    LOCAL CONST Robtarget Tr_meulage_bavure_297 := [[34.2176875,132.965375,122.45971875],[0.142128156611238,-0.169112950759258,-0.746628793402951,0.62749170659495],[0,0,0,0],[8.999999E+09,8.999999E+09,8.999999E+09,8.999999E+09,8.999999E+09,8.999999E+09]];
    LOCAL CONST Robtarget Tr_meulage_bavure_298 := [[35.4824296875,132.352796875,122.428859375],[0.141640226442861,-0.168636903428218,-0.74693783228447,0.62736234805536],[0,0,0,0],[8.999999E+09,8.999999E+09,8.999999E+09,8.999999E+09,8.999999E+09,8.999999E+09]];
    LOCAL CONST Robtarget Tr_meulage_bavure_299 := [[38.3330234375,131.063109375,122.374390625],[0.14118721471856,-0.168181992906434,-0.74720342134066,0.627270304413374],[0,0,0,0],[8.999999E+09,8.999999E+09,8.999999E+09,8.999999E+09,8.999999E+09,8.999999E+09]];
    LOCAL CONST Robtarget Tr_meulage_bavure_300 := [[39.25145703125,130.60725,122.35015625],[0.14084665051928,-0.16784433536859,-0.747410861926925,0.627190165417019],[0,0,0,0],[8.999999E+09,8.999999E+09,8.999999E+09,8.999999E+09,8.999999E+09,8.999999E+09]];
    LOCAL CONST Robtarget Tr_meulage_bavure_301 := [[43.699125,128.5305,122.2544765625],[0.140654971334551,-0.167669079521495,-0.747553059163392,0.627110582390972],[0,0,0,0],[8.999999E+09,8.999999E+09,8.999999E+09,8.999999E+09,8.999999E+09,8.999999E+09]];
    LOCAL CONST Robtarget Tr_meulage_bavure_302 := [[44.1365078125,128.3245625,122.24478125],[0.140603570004533,-0.167647641561045,-0.747634929696438,0.62703023553797],[0,0,0,0],[8.999999E+09,8.999999E+09,8.999999E+09,8.999999E+09,8.999999E+09,8.999999E+09]];
    LOCAL CONST Robtarget Tr_meulage_bavure_303 := [[44.23293359375,128.27996875,122.24278125],[0.14065985839217,-0.167741895489389,-0.747666250712567,0.626955052838826],[0,0,0,0],[8.999999E+09,8.999999E+09,8.999999E+09,8.999999E+09,8.999999E+09,8.999999E+09]];
    LOCAL CONST Robtarget Tr_meulage_bavure_304 := [[44.98623046875,127.9280703125,122.226546875],[0.140804799027706,-0.167930767749504,-0.747654793054834,0.626885616548954],[0,0,0,0],[8.999999E+09,8.999999E+09,8.999999E+09,8.999999E+09,8.999999E+09,8.999999E+09]];
    LOCAL CONST Robtarget Tr_meulage_bavure_305 := [[45.85191015625,127.5197578125,122.20725],[0.141050378042018,-0.168230430617468,-0.747600477109053,0.626814836849593],[0,0,0,0],[8.999999E+09,8.999999E+09,8.999999E+09,8.999999E+09,8.999999E+09,8.999999E+09]];
    LOCAL CONST Robtarget Tr_meulage_bavure_306 := [[46.1492265625,127.3825234375,122.2011171875],[0.141429042259318,-0.168679406784711,-0.747494198232892,0.626735596037544],[0,0,0,0],[8.999999E+09,8.999999E+09,8.999999E+09,8.999999E+09,8.999999E+09,8.999999E+09]];
    LOCAL CONST Robtarget Tr_meulage_bavure_307 := [[46.39677734375,127.2688984375,122.1961171875],[0.14196329956454,-0.16930433923435,-0.747329405658289,0.626642818303695],[0,0,0,0],[8.999999E+09,8.999999E+09,8.999999E+09,8.999999E+09,8.999999E+09,8.999999E+09]];
    LOCAL CONST Robtarget Tr_meulage_bavure_308 := [[46.909359375,127.0229375,122.1839921875],[0.142618884190371,-0.170065666026522,-0.747117380212942,0.62654061583827],[0,0,0,0],[8.999999E+09,8.999999E+09,8.999999E+09,8.999999E+09,8.999999E+09,8.999999E+09]];
    LOCAL CONST Robtarget Tr_meulage_bavure_309 := [[49.37613671875,125.85084375,122.1275625],[0.143287509218809,-0.170833179418583,-0.746885669478168,0.626455514174595],[0,0,0,0],[8.999999E+09,8.999999E+09,8.999999E+09,8.999999E+09,8.999999E+09,8.999999E+09]];
    LOCAL CONST Robtarget Tr_meulage_bavure_310 := [[49.73691796875,125.6805234375,122.1194921875],[0.14380033022182,-0.171406070605532,-0.746681457533514,0.626424955571929],[0,0,0,0],[8.999999E+09,8.999999E+09,8.999999E+09,8.999999E+09,8.999999E+09,8.999999E+09]];
    LOCAL CONST Robtarget Tr_meulage_bavure_311 := [[52.63286328125,124.2019609375,122.0362421875],[0.143984238697923,-0.171578015432722,-0.746552510429731,0.626489323770019],[0,0,0,0],[8.999999E+09,8.999999E+09,8.999999E+09,8.999999E+09,8.999999E+09,8.999999E+09]];
    LOCAL CONST Robtarget Tr_meulage_bavure_312 := [[52.83613671875,124.1022734375,122.031078125],[0.14373566681063,-0.171225947215702,-0.746527398631558,0.62667262280954],[0,0,0,0],[8.999999E+09,8.999999E+09,8.999999E+09,8.999999E+09,8.999999E+09,8.999999E+09]];
    LOCAL CONST Robtarget Tr_meulage_bavure_313 := [[53.12591015625,123.9665546875,122.02478125],[0.143068925856055,-0.170367944227415,-0.746602173269505,0.626969888354593],[0,0,0,0],[8.999999E+09,8.999999E+09,8.999999E+09,8.999999E+09,8.999999E+09,8.999999E+09]];
    LOCAL CONST Robtarget Tr_meulage_bavure_314 := [[54.6938984375,123.250890625,121.99378125],[0.142117463553127,-0.169163701981467,-0.746739221500474,0.627349028498504],[0,0,0,0],[8.999999E+09,8.999999E+09,8.999999E+09,8.999999E+09,8.999999E+09,8.999999E+09]];
    LOCAL CONST Robtarget Tr_meulage_bavure_315 := [[56.9182890625,122.2494375,121.95209375],[0.141085382293744,-0.167857982463528,-0.746884441852941,0.627759701752448],[0,0,0,0],[8.999999E+09,8.999999E+09,8.999999E+09,8.999999E+09,8.999999E+09,8.999999E+09]];
    LOCAL CONST Robtarget Tr_meulage_bavure_316 := [[60.7889375,120.4804609375,121.8751875],[0.140172441622204,-0.166689643799396,-0.746986030179913,0.62815453510721],[0,0,0,0],[8.999999E+09,8.999999E+09,8.999999E+09,8.999999E+09,8.999999E+09,8.999999E+09]];
    LOCAL CONST Robtarget Tr_meulage_bavure_317 := [[61.05184765625,120.35671875,121.8693671875],[0.139514593688367,-0.165820601375903,-0.747009552064025,0.628502931920296],[0,0,0,0],[8.999999E+09,8.999999E+09,8.999999E+09,8.999999E+09,8.999999E+09,8.999999E+09]];
    LOCAL CONST Robtarget Tr_meulage_bavure_318 := [[61.35975390625,120.2146015625,121.8630234375],[0.139157785334625,-0.165307448949311,-0.746948271938196,0.628789978570886],[0,0,0,0],[8.999999E+09,8.999999E+09,8.999999E+09,8.999999E+09,8.999999E+09,8.999999E+09]];
    LOCAL CONST Robtarget Tr_meulage_bavure_319 := [[63.2705546875,119.314625,121.820625],[0.139070684719946,-0.165114117692366,-0.746814191610559,0.629019265205179],[0,0,0,0],[8.999999E+09,8.999999E+09,8.999999E+09,8.999999E+09,8.999999E+09,8.999999E+09]];
    LOCAL CONST Robtarget Tr_meulage_bavure_320 := [[66.2385,117.89525,121.75121875],[0.139180283924146,-0.165155531424716,-0.746630431468063,0.629202270984799],[0,0,0,0],[8.999999E+09,8.999999E+09,8.999999E+09,8.999999E+09,8.999999E+09,8.999999E+09]];
    LOCAL CONST Robtarget Tr_meulage_bavure_321 := [[67.29140625,117.4122578125,121.73],[0.139402451268071,-0.165332948265824,-0.746421577324781,0.629354273602849],[0,0,0,0],[8.999999E+09,8.999999E+09,8.999999E+09,8.999999E+09,8.999999E+09,8.999999E+09]];
    LOCAL CONST Robtarget Tr_meulage_bavure_322 := [[68.7794296875,116.7210546875,121.6985859375],[0.139675077826781,-0.165574350874053,-0.746207051271152,0.629484744533123],[0,0,0,0],[8.999999E+09,8.999999E+09,8.999999E+09,8.999999E+09,8.999999E+09,8.999999E+09]];
    LOCAL CONST Robtarget Tr_meulage_bavure_323 := [[71.4787109375,115.4669375,121.6415625],[0.139968932002636,-0.16584743988122,-0.745998695885669,0.629594528641862],[0,0,0,0],[8.999999E+09,8.999999E+09,8.999999E+09,8.999999E+09,8.999999E+09,8.999999E+09]];
    LOCAL CONST Robtarget Tr_meulage_bavure_324 := [[73.6623046875,114.4688046875,121.598140625],[0.14029056327217,-0.166161157540129,-0.745796819755704,0.629679387644204],[0,0,0,0],[8.999999E+09,8.999999E+09,8.999999E+09,8.999999E+09,8.999999E+09,8.999999E+09]];
    LOCAL CONST Robtarget Tr_meulage_bavure_325 := [[74.165671875,114.234359375,121.5874140625],[0.140681176535999,-0.166565141217583,-0.745591951180769,0.629728118027191],[0,0,0,0],[8.999999E+09,8.999999E+09,8.999999E+09,8.999999E+09,8.999999E+09,8.999999E+09]];
    LOCAL CONST Robtarget Tr_meulage_bavure_326 := [[74.6225,114.02121875,121.5776171875],[0.141192737880537,-0.167122613384322,-0.745373159529928,0.629724936712661],[0,0,0,0],[8.999999E+09,8.999999E+09,8.999999E+09,8.999999E+09,8.999999E+09,8.999999E+09]];
    LOCAL CONST Robtarget Tr_meulage_bavure_327 := [[75.4216484375,113.656734375,121.561859375],[0.141859319446395,-0.167873698675355,-0.745130708530274,0.629662276132558],[0,0,0,0],[8.999999E+09,8.999999E+09,8.999999E+09,8.999999E+09,8.999999E+09,8.999999E+09]];
    LOCAL CONST Robtarget Tr_meulage_bavure_328 := [[78.572046875,112.1458046875,121.48746875],[0.14266757437261,-0.168803513747482,-0.744869090570777,0.629540606221238],[0,0,0,0],[8.999999E+09,8.999999E+09,8.999999E+09,8.999999E+09,8.999999E+09,8.999999E+09]];
    LOCAL CONST Robtarget Tr_meulage_bavure_329 := [[79.279515625,111.8110390625,121.471515625],[0.143538630388157,-0.169818250402327,-0.744607856091829,0.629378712750054],[0,0,0,0],[8.999999E+09,8.999999E+09,8.999999E+09,8.999999E+09,8.999999E+09,8.999999E+09]];
    LOCAL CONST Robtarget Tr_meulage_bavure_330 := [[79.8409140625,111.541390625,121.4581953125],[0.144333710343636,-0.170752769943249,-0.744382392618626,0.629210716035985],[0,0,0,0],[8.999999E+09,8.999999E+09,8.999999E+09,8.999999E+09,8.999999E+09,8.999999E+09]];
    LOCAL CONST Robtarget Tr_meulage_bavure_331 := [[81.0044375,110.971453125,121.42875],[0.144890710586549,-0.171415587872169,-0.744237400404596,0.629073978208583],[0,0,0,0],[8.999999E+09,8.999999E+09,8.999999E+09,8.999999E+09,8.999999E+09,8.999999E+09]];
    LOCAL CONST Robtarget Tr_meulage_bavure_332 := [[82.0306171875,110.47190625,121.4032890625],[0.14507897492011,-0.171650738096502,-0.74420683512921,0.62900262455257],[0,0,0,0],[8.999999E+09,8.999999E+09,8.999999E+09,8.999999E+09,8.999999E+09,8.999999E+09]];
    LOCAL CONST Robtarget Tr_meulage_bavure_333 := [[82.2463984375,110.37040625,121.3985234375],[0.144848305949184,-0.171396979313194,-0.744301822780907,0.629012591567915],[0,0,0,0],[8.999999E+09,8.999999E+09,8.999999E+09,8.999999E+09,8.999999E+09,8.999999E+09]];
    LOCAL CONST Robtarget Tr_meulage_bavure_334 := [[82.8360078125,110.102390625,121.387046875],[0.144249846582567,-0.170713885772361,-0.744506711868629,0.629093400814195],[0,0,0,0],[8.999999E+09,8.999999E+09,8.999999E+09,8.999999E+09,8.999999E+09,8.999999E+09]];
    LOCAL CONST Robtarget Tr_meulage_bavure_335 := [[87.9835546875,107.8033984375,121.2936484375],[0.143422785192236,-0.169764675381047,-0.744780598167888,0.629215162144995],[0,0,0,0],[8.999999E+09,8.999999E+09,8.999999E+09,8.999999E+09,8.999999E+09,8.999999E+09]];
    LOCAL CONST Robtarget Tr_meulage_bavure_336 := [[89.505015625,107.101125,121.2622734375],[0.142553575426364,-0.168768800133135,-0.745070641436071,0.629337198570706],[0,0,0,0],[8.999999E+09,8.999999E+09,8.999999E+09,8.999999E+09,8.999999E+09,8.999999E+09]];
    LOCAL CONST Robtarget Tr_meulage_bavure_337 := [[90.2310703125,106.7596171875,121.2462421875],[0.14182660803926,-0.167943707343211,-0.745326103780332,0.629419671951494],[0,0,0,0],[8.999999E+09,8.999999E+09,8.999999E+09,8.999999E+09,8.999999E+09,8.999999E+09]];
    LOCAL CONST Robtarget Tr_meulage_bavure_338 := [[90.8233671875,106.4939140625,121.235296875],[0.141376345637687,-0.167449055194185,-0.745512389605452,0.629432140705792],[0,0,0,0],[8.999999E+09,8.999999E+09,8.999999E+09,8.999999E+09,8.999999E+09,8.999999E+09]];
    LOCAL CONST Robtarget Tr_meulage_bavure_339 := [[94.6694375,104.71,121.1545390625],[0.141264646733224,-0.167358108160957,-0.745613339390501,0.629361828632043],[0,0,0,0],[8.999999E+09,8.999999E+09,8.999999E+09,8.999999E+09,8.999999E+09,8.999999E+09]];
    LOCAL CONST Robtarget Tr_meulage_bavure_340 := [[95.751984375,104.22146875,121.1340625],[0.141467329288269,-0.167642452943014,-0.745635426500155,0.629214441556474],[0,0,0,0],[8.999999E+09,8.999999E+09,8.999999E+09,8.999999E+09,8.999999E+09,8.999999E+09]];
    LOCAL CONST Robtarget Tr_meulage_bavure_341 := [[96.68790625,103.7821953125,121.1135546875],[0.141877475777199,-0.168176984297917,-0.745609015898498,0.629010714718296],[0,0,0,0],[8.999999E+09,8.999999E+09,8.999999E+09,8.999999E+09,8.999999E+09,8.999999E+09]];
    LOCAL CONST Robtarget Tr_meulage_bavure_342 := [[97.9893046875,103.179171875,121.086328125],[0.142335202704554,-0.168773211692481,-0.745577870908683,0.628784487322432],[0,0,0,0],[8.999999E+09,8.999999E+09,8.999999E+09,8.999999E+09,8.999999E+09,8.999999E+09]];
    LOCAL CONST Robtarget Tr_meulage_bavure_343 := [[98.1599609375,103.097578125,121.08234375],[0.142668858237759,-0.169228047714292,-0.745588756710536,0.628573679549805],[0,0,0,0],[8.999999E+09,8.999999E+09,8.999999E+09,8.999999E+09,8.999999E+09,8.999999E+09]];
    LOCAL CONST Robtarget Tr_meulage_bavure_344 := [[101.117515625,101.6851328125,121.0135],[0.142745339161701,-0.169384774528264,-0.745680109312349,0.62840571359715],[0,0,0,0],[8.999999E+09,8.999999E+09,8.999999E+09,8.999999E+09,8.999999E+09,8.999999E+09]];
    LOCAL CONST Robtarget Tr_meulage_bavure_345 := [[101.7760234375,101.3719765625,120.998390625],[0.142507331671173,-0.169175652200885,-0.745868675580983,0.628292271088415],[0,0,0,0],[8.999999E+09,8.999999E+09,8.999999E+09,8.999999E+09,8.999999E+09,8.999999E+09]];
    LOCAL CONST Robtarget Tr_meulage_bavure_346 := [[105.635125,99.6135,120.922578125],[0.141982136855868,-0.168632638895959,-0.746146933528534,0.628226758025152],[0,0,0,0],[8.999999E+09,8.999999E+09,8.999999E+09,8.999999E+09,8.999999E+09,8.999999E+09]];
    LOCAL CONST Robtarget Tr_meulage_bavure_347 := [[106.666,99.137140625,120.901234375],[0.141275871200478,-0.167879804158259,-0.746483307089515,0.628188006737658],[0,0,0,0],[8.999999E+09,8.999999E+09,8.999999E+09,8.999999E+09,8.999999E+09,8.999999E+09]];
    LOCAL CONST Robtarget Tr_meulage_bavure_348 := [[106.8926953125,99.0316953125,120.896421875],[0.140531773528285,-0.16708577567627,-0.746836906802689,0.628146319604792],[0,0,0,0],[8.999999E+09,8.999999E+09,8.999999E+09,8.999999E+09,8.999999E+09,8.999999E+09]];
    LOCAL CONST Robtarget Tr_meulage_bavure_349 := [[110.709515625,97.2290859375,120.8109296875],[0.139903160526474,-0.166430816633961,-0.747163563506302,0.628072048667843],[0,0,0,0],[8.999999E+09,8.999999E+09,8.999999E+09,8.999999E+09,8.999999E+09,8.999999E+09]];
    LOCAL CONST Robtarget Tr_meulage_bavure_350 := [[114.4970078125,95.529703125,120.7409140625],[0.139533545167416,-0.1660823922192,-0.747419536379912,0.62794192837029],[0,0,0,0],[8.999999E+09,8.999999E+09,8.999999E+09,8.999999E+09,8.999999E+09,8.999999E+09]];
    LOCAL CONST Robtarget Tr_meulage_bavure_351 := [[114.5951640625,95.4851484375,120.739015625],[0.13953408653618,-0.16616858354886,-0.74756747143012,0.627742874268961],[0,0,0,0],[8.999999E+09,8.999999E+09,8.999999E+09,8.999999E+09,8.999999E+09,8.999999E+09]];
    LOCAL CONST Robtarget Tr_meulage_bavure_352 := [[114.637203125,95.4663359375,120.7382421875],[0.13997290600938,-0.166765691405124,-0.747579507661621,0.627472445194105],[0,0,0,0],[8.999999E+09,8.999999E+09,8.999999E+09,8.999999E+09,8.999999E+09,8.999999E+09]];
    LOCAL CONST Robtarget Tr_meulage_bavure_353 := [[118.0484765625,93.8467421875,120.660421875],[0.140853009814362,-0.167871748403136,-0.74744303644807,0.627143056231669],[0,0,0,0],[8.999999E+09,8.999999E+09,8.999999E+09,8.999999E+09,8.999999E+09,8.999999E+09]];
    LOCAL CONST Robtarget Tr_meulage_bavure_354 := [[118.5088671875,93.5909453125,120.64375],[0.142108776667301,-0.169401922842107,-0.747161945454812,0.626783145430459],[0,0,0,0],[8.999999E+09,8.999999E+09,8.999999E+09,8.999999E+09,8.999999E+09,8.999999E+09]];
    LOCAL CONST Robtarget Tr_meulage_bavure_355 := [[119.5866875,93.05265625,120.6147578125],[0.143616222822991,-0.171201177424273,-0.746756071337723,0.626434280121106],[0,0,0,0],[8.999999E+09,8.999999E+09,8.999999E+09,8.999999E+09,8.999999E+09,8.999999E+09]];
    LOCAL CONST Robtarget Tr_meulage_bavure_356 := [[121.79125,92.0239296875,120.5674453125],[0.145225138008046,-0.173081765686502,-0.746252321487508,0.626146815333187],[0,0,0,0],[8.999999E+09,8.999999E+09,8.999999E+09,8.999999E+09,8.999999E+09,8.999999E+09]];
    LOCAL CONST Robtarget Tr_meulage_bavure_357 := [[122.4661953125,91.7112890625,120.5533359375],[0.146804469278541,-0.174878619242286,-0.745674508908111,0.625967605468849],[0,0,0,0],[8.999999E+09,8.999999E+09,8.999999E+09,8.999999E+09,8.999999E+09,8.999999E+09]];
    LOCAL CONST Robtarget Tr_meulage_bavure_358 := [[123.41609375,91.2462734375,120.52934375],[0.148269237216507,-0.176482035462568,-0.745035857203988,0.625932820624181],[0,0,0,0],[8.999999E+09,8.999999E+09,8.999999E+09,8.999999E+09,8.999999E+09,8.999999E+09]];
    LOCAL CONST Robtarget Tr_meulage_bavure_359 := [[124.916078125,90.4808125,120.4862890625],[0.149574585438793,-0.177831480392815,-0.744340790176818,0.626067245630262],[0,0,0,0],[8.999999E+09,8.999999E+09,8.999999E+09,8.999999E+09,8.999999E+09,8.999999E+09]];
    LOCAL CONST Robtarget Tr_meulage_bavure_360 := [[125.2375078125,90.351828125,120.4828671875],[0.150696883983553,-0.178892913803661,-0.743589020126342,0.626388971563221],[0,0,0,0],[8.999999E+09,8.999999E+09,8.999999E+09,8.999999E+09,8.999999E+09,8.999999E+09]];
    LOCAL CONST Robtarget Tr_meulage_bavure_361 := [[130.249375,87.7945625,120.3390625],[0.151600109700444,-0.17961762579984,-0.742782579183434,0.626920214463091],[0,0,0,0],[8.999999E+09,8.999999E+09,8.999999E+09,8.999999E+09,8.999999E+09,8.999999E+09]];
    LOCAL CONST Robtarget Tr_meulage_bavure_362 := [[130.609796875,87.602,120.3272890625],[0.152230571198168,-0.179938290147757,-0.741930174130846,0.627684380597091],[0,0,0,0],[8.999999E+09,8.999999E+09,8.999999E+09,8.999999E+09,8.999999E+09,8.999999E+09]];
    LOCAL CONST Robtarget Tr_meulage_bavure_363 := [[130.771234375,87.5274765625,120.323953125],[0.152526036565618,-0.179780585465442,-0.741044667303266,0.628703070074163],[0,0,0,0],[8.999999E+09,8.999999E+09,8.999999E+09,8.999999E+09,8.999999E+09,8.999999E+09]];
    LOCAL CONST Robtarget Tr_meulage_bavure_364 := [[131.62240625,87.1239140625,120.3046328125],[0.152438548541072,-0.179091243284413,-0.740137244094725,0.629988631168373],[0,0,0,0],[8.999999E+09,8.999999E+09,8.999999E+09,8.999999E+09,8.999999E+09,8.999999E+09]];
    LOCAL CONST Robtarget Tr_meulage_bavure_365 := [[132.93284375,86.4797578125,120.2710859375],[0.151956809779417,-0.177859085261569,-0.739202461606242,0.631549676990537],[0,0,0,0],[8.999999E+09,8.999999E+09,8.999999E+09,8.999999E+09,8.999999E+09,8.999999E+09]];
    LOCAL CONST Robtarget Tr_meulage_bavure_366 := [[135.80690625,85.059875,120.19634375],[0.151096320751359,-0.176108478208518,-0.738230061565139,0.633381466385],[0,0,0,0],[8.999999E+09,8.999999E+09,8.999999E+09,8.999999E+09,8.999999E+09,8.999999E+09]];
    LOCAL CONST Robtarget Tr_meulage_bavure_367 := [[136.79134375,84.576375,120.17121875],[0.149940500700765,-0.173945899218158,-0.737193751145513,0.63545734999825],[0,0,0,0],[8.999999E+09,8.999999E+09,8.999999E+09,8.999999E+09,8.999999E+09,8.999999E+09]];
    LOCAL CONST Robtarget Tr_meulage_bavure_368 := [[136.829109375,84.5587265625,120.17040625],[0.148641429765737,-0.171556234855416,-0.736049162251626,0.637734909181009],[0,0,0,0],[8.999999E+09,8.999999E+09,8.999999E+09,8.999999E+09,8.999999E+09,8.999999E+09]];
    LOCAL CONST Robtarget Tr_meulage_bavure_369 := [[137.133640625,84.42059375,120.1645234375],[0.147464120430556,-0.169249901817863,-0.73472270026981,0.640149480690663],[0,0,0,0],[8.999999E+09,8.999999E+09,8.999999E+09,8.999999E+09,8.999999E+09,8.999999E+09]];
    LOCAL CONST Robtarget Tr_meulage_bavure_370 := [[140.63628125,82.8104609375,120.0933828125],[0.146986350486515,-0.167690776837463,-0.733070237740176,0.642559602429117],[0,0,0,0],[8.999999E+09,8.999999E+09,8.999999E+09,8.999999E+09,8.999999E+09,8.999999E+09]];
    LOCAL CONST Robtarget Tr_meulage_bavure_371 := [[141.266359375,82.5186875,120.0802265625],[0.148142391817507,-0.167930068945617,-0.730862472645966,0.644742871048865],[0,0,0,0],[8.999999E+09,8.999999E+09,8.999999E+09,8.999999E+09,8.999999E+09,8.999999E+09]];
    LOCAL CONST Robtarget Tr_meulage_bavure_372 := [[142.5813125,81.880578125,120.0479453125],[0.152434602161972,-0.171629578574627,-0.727714383484515,0.646327127615551],[0,0,0,0],[8.999999E+09,8.999999E+09,8.999999E+09,8.999999E+09,8.999999E+09,8.999999E+09]];
    LOCAL CONST Robtarget Tr_meulage_bavure_373 := [[144.158984375,81.1890390625,120.021484375],[0.162044669466051,-0.181158364938845,-0.72298100893018,0.646700574173721],[0,0,0,0],[8.999999E+09,8.999999E+09,8.999999E+09,8.999999E+09,8.999999E+09,8.999999E+09]];
    LOCAL CONST Robtarget Tr_meulage_bavure_374 := [[145.088796875,80.759390625,120.002234375],[0.179704355427492,-0.199423076530988,-0.715612269781922,0.644853363583436],[0,0,0,0],[8.999999E+09,8.999999E+09,8.999999E+09,8.999999E+09,8.999999E+09,8.999999E+09]];
    LOCAL CONST Robtarget Tr_meulage_bavure_375 := [[145.703890625,80.348546875,119.9685],[0.20826350300746,-0.229366043937516,-0.703917224255588,0.639154185310418],[0,0,0,0],[8.999999E+09,8.999999E+09,8.999999E+09,8.999999E+09,8.999999E+09,8.999999E+09]];
    LOCAL CONST Robtarget Tr_meulage_bavure_376 := [[146.073796875,80.104765625,119.9487578125],[0.249501908876202,-0.272659142252544,-0.685506214756904,0.627285436737455],[0,0,0,0],[8.999999E+09,8.999999E+09,8.999999E+09,8.999999E+09,8.999999E+09,8.999999E+09]];
    LOCAL CONST Robtarget Tr_meulage_bavure_377 := [[146.36646875,79.8232265625,119.9184453125],[0.302195458500763,-0.327663362829496,-0.658031174941505,0.60688516073956],[0,0,0,0],[8.999999E+09,8.999999E+09,8.999999E+09,8.999999E+09,8.999999E+09,8.999999E+09]];
    LOCAL CONST Robtarget Tr_meulage_bavure_378 := [[146.751390625,79.510375,119.88809375],[0.360532341612847,-0.387859847783662,-0.621313986745368,0.577537963256935],[0,0,0,0],[8.999999E+09,8.999999E+09,8.999999E+09,8.999999E+09,8.999999E+09,8.999999E+09]];
    LOCAL CONST Robtarget Tr_meulage_bavure_379 := [[147.11709375,78.843578125,119.7979765625],[0.416103296088596,-0.444175563256471,-0.579055221322691,0.542458446932972],[0,0,0,0],[8.999999E+09,8.999999E+09,8.999999E+09,8.999999E+09,8.999999E+09,8.999999E+09]];
    LOCAL CONST Robtarget Tr_meulage_bavure_380 := [[147.616875,77.9455546875,119.677015625],[0.462807025219069,-0.490281336351501,-0.537053900293808,0.506958555320326],[0,0,0,0],[8.999999E+09,8.999999E+09,8.999999E+09,8.999999E+09,8.999999E+09,8.999999E+09]];
    LOCAL CONST Robtarget Tr_meulage_bavure_381 := [[147.638296875,77.7655390625,119.6483671875],[0.499078740896148,-0.52481979087935,-0.499688445924563,0.475180023250522],[0,0,0,0],[8.999999E+09,8.999999E+09,8.999999E+09,8.999999E+09,8.999999E+09,8.999999E+09]];
    LOCAL CONST Robtarget Tr_meulage_bavure_382 := [[147.771859375,76.6325859375,119.467984375],[0.526153881956454,-0.549399765419487,-0.468788601787221,0.448953491013879],[0,0,0,0],[8.999999E+09,8.999999E+09,8.999999E+09,8.999999E+09,8.999999E+09,8.999999E+09]];
    LOCAL CONST Robtarget Tr_meulage_bavure_383 := [[147.711265625,75.7255859375,119.3142109375],[0.545968775974128,-0.566305336226663,-0.444495132259534,0.428532891643217],[0,0,0,0],[8.999999E+09,8.999999E+09,8.999999E+09,8.999999E+09,8.999999E+09,8.999999E+09]];
    LOCAL CONST Robtarget Tr_meulage_bavure_384 := [[147.602359375,75.4485078125,119.2621796875],[0.560232306595868,-0.577501822390566,-0.42622413873022,0.413478404932509],[0,0,0,0],[8.999999E+09,8.999999E+09,8.999999E+09,8.999999E+09,8.999999E+09,8.999999E+09]];
    LOCAL CONST Robtarget Tr_meulage_bavure_385 := [[147.353203125,73.9746953125,119.0038828125],[0.570335925633924,-0.584569685115412,-0.413038763251024,0.402981631377198],[0,0,0,0],[8.999999E+09,8.999999E+09,8.999999E+09,8.999999E+09,8.999999E+09,8.999999E+09]];
    LOCAL CONST Robtarget Tr_meulage_bavure_386 := [[147.056203125,73.1938828125,118.8578125],[0.577428113316374,-0.588783928814792,-0.403819158256316,0.396030739395909],[0,0,0,0],[8.999999E+09,8.999999E+09,8.999999E+09,8.999999E+09,8.999999E+09,8.999999E+09]];
    LOCAL CONST Robtarget Tr_meulage_bavure_387 := [[146.640046875,72.1850234375,118.667265625],[0.582486218866137,-0.591207337188674,-0.397371317914441,0.39150954647907],[0,0,0,0],[8.999999E+09,8.999999E+09,8.999999E+09,8.999999E+09,8.999999E+09,8.999999E+09]];
    LOCAL CONST Robtarget Tr_meulage_bavure_388 := [[146.107890625,70.7783046875,118.4042734375],[0.586291892586572,-0.592664157602932,-0.392624559613658,0.388403100101227],[0,0,0,0],[8.999999E+09,8.999999E+09,8.999999E+09,8.999999E+09,8.999999E+09,8.999999E+09]];
    LOCAL CONST Robtarget Tr_meulage_bavure_389 := [[145.91209375,70.4478125,118.3385234375],[0.589348182020745,-0.593666695185621,-0.388857604432012,0.386028935251779],[0,0,0,0],[8.999999E+09,8.999999E+09,8.999999E+09,8.999999E+09,8.999999E+09,8.999999E+09]];
    LOCAL CONST Robtarget Tr_meulage_bavure_390 := [[145.85253125,70.3119375,118.3126640625],[0.591897212754762,-0.594456970483624,-0.385718248964095,0.384057329304687],[0,0,0,0],[8.999999E+09,8.999999E+09,8.999999E+09,8.999999E+09,8.999999E+09,8.999999E+09]];
    LOCAL CONST Robtarget Tr_meulage_bavure_391 := [[145.6580625,69.9100859375,118.2351640625],[0.59400517306223,-0.595081099755775,-0.383123111829349,0.382430412324861],[0,0,0,0],[8.999999E+09,8.999999E+09,8.999999E+09,8.999999E+09,8.999999E+09,8.999999E+09]];
    LOCAL CONST Robtarget Tr_meulage_bavure_392 := [[145.122125,68.739765625,118.0111484375],[0.595670947769008,-0.595512083705692,-0.381093153357091,0.38119481713269],[0,0,0,0],[8.999999E+09,8.999999E+09,8.999999E+09,8.999999E+09,8.999999E+09,8.999999E+09]];
    LOCAL CONST Robtarget Tr_meulage_bavure_393 := [[144.237578125,66.7826640625,117.6371953125],[0.596908321308949,-0.595733368588404,-0.379626904027464,0.380375634394434],[0,0,0,0],[8.999999E+09,8.999999E+09,8.999999E+09,8.999999E+09,8.999999E+09,8.999999E+09]];
    LOCAL CONST Robtarget Tr_meulage_bavure_394 := [[143.894546875,65.983515625,117.485515625],[0.59781976996364,-0.595811294891798,-0.378584529254396,0.379860734650486],[0,0,0,0],[8.999999E+09,8.999999E+09,8.999999E+09,8.999999E+09,8.999999E+09,8.999999E+09]];
    LOCAL CONST Robtarget Tr_meulage_bavure_395 := [[143.771640625,65.7254921875,117.435859375],[0.598575401989977,-0.595877689391033,-0.377718489187417,0.379428531273699],[0,0,0,0],[8.999999E+09,8.999999E+09,8.999999E+09,8.999999E+09,8.999999E+09,8.999999E+09]];
    LOCAL CONST Robtarget Tr_meulage_bavure_396 := [[143.505390625,65.138359375,117.323625],[0.599349117415602,-0.596068776879129,-0.376773059900974,0.378846552070645],[0,0,0,0],[8.999999E+09,8.999999E+09,8.999999E+09,8.999999E+09,8.999999E+09,8.999999E+09]];
    LOCAL CONST Robtarget Tr_meulage_bavure_397 := [[142.287015625,62.731515625,116.8564296875],[0.600243844248007,-0.596454499585234,-0.375600269184009,0.377986501287813],[0,0,0,0],[8.999999E+09,8.999999E+09,8.999999E+09,8.999999E+09,8.999999E+09,8.999999E+09]];
    LOCAL CONST Robtarget Tr_meulage_bavure_398 := [[140.7463125,59.19300390625,116.1835859375],[0.601238686033111,-0.596982227985233,-0.374245840806582,0.376914197830144],[0,0,0,0],[8.999999E+09,8.999999E+09,8.999999E+09,8.999999E+09,8.999999E+09,8.999999E+09]];
    LOCAL CONST Robtarget Tr_meulage_bavure_399 := [[140.450890625,58.5961484375,116.0681015625],[0.602192204492973,-0.597486547384532,-0.372944305569855,0.375881523203022],[0,0,0,0],[8.999999E+09,8.999999E+09,8.999999E+09,8.999999E+09,8.999999E+09,8.999999E+09]];
    LOCAL CONST Robtarget Tr_meulage_bavure_400 := [[140.00378125,57.6006328125,115.8780390625],[0.602906871593234,-0.597757325053511,-0.372017935530549,0.375222787386534],[0,0,0,0],[8.999999E+09,8.999999E+09,8.999999E+09,8.999999E+09,8.999999E+09,8.999999E+09]];
    LOCAL CONST Robtarget Tr_meulage_bavure_401 := [[139.5975625,56.73630078125,115.712015625],[0.603226087226463,-0.59762548637184,-0.371725734629334,0.375209333496058],[0,0,0,0],[8.999999E+09,8.999999E+09,8.999999E+09,8.999999E+09,8.999999E+09,8.999999E+09]];
    LOCAL CONST Robtarget Tr_meulage_bavure_402 := [[138.86434375,55.33035546875,115.43790625],[0.603103449797866,-0.597040205189456,-0.372143820708253,0.375923129027609],[0,0,0,0],[8.999999E+09,8.999999E+09,8.999999E+09,8.999999E+09,8.999999E+09,8.999999E+09]];
    LOCAL CONST Robtarget Tr_meulage_bavure_403 := [[137.97534375,53.60463671875,115.1020703125],[0.602614330047082,-0.596082147278622,-0.373144516718151,0.377233631269525],[0,0,0,0],[8.999999E+09,8.999999E+09,8.999999E+09,8.999999E+09,8.999999E+09,8.999999E+09]];
    LOCAL CONST Robtarget Tr_meulage_bavure_404 := [[137.442171875,52.35215234375,114.8645859375],[0.601923377714026,-0.594923432309849,-0.374456477629714,0.378862380569982],[0,0,0,0],[8.999999E+09,8.999999E+09,8.999999E+09,8.999999E+09,8.999999E+09,8.999999E+09]];
    LOCAL CONST Robtarget Tr_meulage_bavure_405 := [[137.19253125,51.788625,114.7571953125],[0.601219547195672,-0.593760706474136,-0.375774740719548,0.380495234864147],[0,0,0,0],[8.999999E+09,8.999999E+09,8.999999E+09,8.999999E+09,8.999999E+09,8.999999E+09]];
    LOCAL CONST Robtarget Tr_meulage_bavure_406 := [[136.576234375,50.4181171875,114.4955],[0.600658656084442,-0.592758369730777,-0.376852647312035,0.381875341176744],[0,0,0,0],[8.999999E+09,8.999999E+09,8.999999E+09,8.999999E+09,8.999999E+09,8.999999E+09]];
    LOCAL CONST Robtarget Tr_meulage_bavure_407 := [[136.09378125,49.38021484375,114.2964296875],[0.600334430615642,-0.592031545332389,-0.377538894832942,0.382833650084547],[0,0,0,0],[8.999999E+09,8.999999E+09,8.999999E+09,8.999999E+09,8.999999E+09,8.999999E+09]];
    LOCAL CONST Robtarget Tr_meulage_bavure_408 := [[135.309703125,47.78010546875,113.98728125],[0.600287884328917,-0.591637778793676,-0.377766949819651,0.38329013326194],[0,0,0,0],[8.999999E+09,8.999999E+09,8.999999E+09,8.999999E+09,8.999999E+09,8.999999E+09]];
    LOCAL CONST Robtarget Tr_meulage_bavure_409 := [[134.64565625,46.4082109375,113.7226875],[0.600521544077413,-0.591591025739444,-0.377530317372852,0.38322942583756],[0,0,0,0],[8.999999E+09,8.999999E+09,8.999999E+09,8.999999E+09,8.999999E+09,8.999999E+09]];
    LOCAL CONST Robtarget Tr_meulage_bavure_410 := [[133.51640625,43.938890625,113.250125],[0.600991084014193,-0.591863687584454,-0.376890035023714,0.382702225959297],[0,0,0,0],[8.999999E+09,8.999999E+09,8.999999E+09,8.999999E+09,8.999999E+09,8.999999E+09]];
    LOCAL CONST Robtarget Tr_meulage_bavure_411 := [[133.511625,43.928171875,113.248078125],[0.601615816288487,-0.592385008932363,-0.37596472459449,0.381823174577356],[0,0,0,0],[8.999999E+09,8.999999E+09,8.999999E+09,8.999999E+09,8.999999E+09,8.999999E+09]];
    LOCAL CONST Robtarget Tr_meulage_bavure_412 := [[133.510015625,43.92501171875,113.2474609375],[0.602275613687394,-0.593042842234446,-0.374935378302141,0.380772549600668],[0,0,0,0],[8.999999E+09,8.999999E+09,8.999999E+09,8.999999E+09,8.999999E+09,8.999999E+09]];
    LOCAL CONST Robtarget Tr_meulage_bavure_413 := [[131.404375,39.44476171875,112.3868828125],[0.602823048327336,-0.593694375880212,-0.374029495524725,0.37978059051387],[0,0,0,0],[8.999999E+09,8.999999E+09,8.999999E+09,8.999999E+09,8.999999E+09,8.999999E+09]];
    LOCAL CONST Robtarget Tr_meulage_bavure_414 := [[131.35328125,39.33466015625,112.365765625],[0.603125994869896,-0.594205559379643,-0.373456695332266,0.379063166538279],[0,0,0,0],[8.999999E+09,8.999999E+09,8.999999E+09,8.999999E+09,8.999999E+09,8.999999E+09]];
    LOCAL CONST Robtarget Tr_meulage_bavure_415 := [[131.2973125,39.220609375,112.3437265625],[0.603099379066155,-0.594485902063001,-0.373355747014302,0.378765280074284],[0,0,0,0],[8.999999E+09,8.999999E+09,8.999999E+09,8.999999E+09,8.999999E+09,8.999999E+09]];
    LOCAL CONST Robtarget Tr_meulage_bavure_416 := [[130.133390625,36.91419921875,111.896234375],[0.602742640901433,-0.594520016245346,-0.373735763076247,0.37890478819964],[0,0,0,0],[8.999999E+09,8.999999E+09,8.999999E+09,8.999999E+09,8.999999E+09,8.999999E+09]];
    LOCAL CONST Robtarget Tr_meulage_bavure_417 := [[129.9936484375,36.67788671875,111.8492421875],[0.60214414923868,-0.594373862084521,-0.374467492630725,0.379362929885374],[0,0,0,0],[8.999999E+09,8.999999E+09,8.999999E+09,8.999999E+09,8.999999E+09,8.999999E+09]];
    LOCAL CONST Robtarget Tr_meulage_bavure_418 := [[128.9553515625,34.442203125,111.4205],[0.601447466675635,-0.594173105220638,-0.37533235143633,0.379927482326826],[0,0,0,0],[8.999999E+09,8.999999E+09,8.999999E+09,8.999999E+09,8.999999E+09,8.999999E+09]];
    LOCAL CONST Robtarget Tr_meulage_bavure_419 := [[127.6177421875,31.6041484375,110.875140625],[0.600803332550347,-0.594046077705111,-0.376103867569437,0.380382036850957],[0,0,0,0],[8.999999E+09,8.999999E+09,8.999999E+09,8.999999E+09,8.999999E+09,8.999999E+09]];
    LOCAL CONST Robtarget Tr_meulage_bavure_420 := [[127.4825703125,31.3023203125,110.8175390625],[0.600308454877326,-0.594070631718676,-0.376639851356928,0.380594621483281],[0,0,0,0],[8.999999E+09,8.999999E+09,8.999999E+09,8.999999E+09,8.999999E+09,8.999999E+09]];
    LOCAL CONST Robtarget Tr_meulage_bavure_421 := [[126.9286953125,30.173580078125,110.599421875],[0.599976001596739,-0.594236846970697,-0.376930862672717,0.380571270559293],[0,0,0,0],[8.999999E+09,8.999999E+09,8.999999E+09,8.999999E+09,8.999999E+09,8.999999E+09]];
    LOCAL CONST Robtarget Tr_meulage_bavure_422 := [[125.4919140625,27.304275390625,110.0433359375],[0.599742995286528,-0.594463550928519,-0.377083933072169,0.380432824084653],[0,0,0,0],[8.999999E+09,8.999999E+09,8.999999E+09,8.999999E+09,8.999999E+09,8.999999E+09]];
    LOCAL CONST Robtarget Tr_meulage_bavure_423 := [[124.0481171875,24.3710234375,109.476265625],[0.599513522819978,-0.59464386905713,-0.377254340414251,0.380343749241861],[0,0,0,0],[8.999999E+09,8.999999E+09,8.999999E+09,8.999999E+09,8.999999E+09,8.999999E+09]];
    LOCAL CONST Robtarget Tr_meulage_bavure_424 := [[123.800125,23.872529296875,109.3797421875],[0.599220692677942,-0.594697609671078,-0.377553137296733,0.380424687731314],[0,0,0,0],[8.999999E+09,8.999999E+09,8.999999E+09,8.999999E+09,8.999999E+09,8.999999E+09]];
    LOCAL CONST Robtarget Tr_meulage_bavure_425 := [[123.7095859375,23.692724609375,109.3448671875],[0.598866257997872,-0.594617075914202,-0.377981823080886,0.380682911992803],[0,0,0,0],[8.999999E+09,8.999999E+09,8.999999E+09,8.999999E+09,8.999999E+09,8.999999E+09]];
    LOCAL CONST Robtarget Tr_meulage_bavure_426 := [[122.650984375,21.4718828125,108.917453125],[0.598527332921101,-0.594475570958536,-0.378421145074746,0.381000346771751],[0,0,0,0],[8.999999E+09,8.999999E+09,8.999999E+09,8.999999E+09,8.999999E+09,8.999999E+09]];
    LOCAL CONST Robtarget Tr_meulage_bavure_427 := [[122.290046875,20.6795078125,108.765890625],[0.598382537232284,-0.594446198080771,-0.378594439867025,0.381101439021877],[0,0,0,0],[8.999999E+09,8.999999E+09,8.999999E+09,8.999999E+09,8.999999E+09,8.999999E+09]];
    LOCAL CONST Robtarget Tr_meulage_bavure_428 := [[121.7777734375,19.671919921875,108.5701875],[0.598791531276182,-0.594890600864877,-0.377938125889626,0.380416414043332],[0,0,0,0],[8.999999E+09,8.999999E+09,8.999999E+09,8.999999E+09,8.999999E+09,8.999999E+09]];
    LOCAL CONST Robtarget Tr_meulage_bavure_429 := [[120.432734375,17.050373046875,108.0603125],[0.600512988647233,-0.596566672719918,-0.375248746188613,0.377731033871627],[0,0,0,0],[8.999999E+09,8.999999E+09,8.999999E+09,8.999999E+09,8.999999E+09,8.999999E+09]];
    LOCAL CONST Robtarget Tr_meulage_bavure_430 := [[119.6466875,15.1556005859375,107.702203125],[0.604661126658193,-0.600586385294265,-0.368666785561249,0.371168044060301],[0,0,0,0],[8.999999E+09,8.999999E+09,8.999999E+09,8.999999E+09,8.999999E+09,8.999999E+09]];
    LOCAL CONST Robtarget Tr_meulage_bavure_431 := [[119.5239296875,14.882251953125,107.650015625],[0.610211808403804,-0.605942062354134,-0.359615628534783,0.362149645406579],[0,0,0,0],[8.999999E+09,8.999999E+09,8.999999E+09,8.999999E+09,8.999999E+09,8.999999E+09]];
    LOCAL CONST Robtarget Tr_meulage_bavure_432 := [[119.2741640625,14.3379033203125,107.5457890625],[0.612261014665673,-0.607771290583205,-0.356278127194006,0.358910022633135],[0,0,0,0],[8.999999E+09,8.999999E+09,8.999999E+09,8.999999E+09,8.999999E+09,8.999999E+09]];
    LOCAL CONST Robtarget Tr_meulage_bavure_433 := [[118.5250546875,12.7655537109375,107.243203125],[0.610505912012204,-0.605789044185102,-0.359362810810891,0.36216092493468],[0,0,0,0],[8.999999E+09,8.999999E+09,8.999999E+09,8.999999E+09,8.999999E+09,8.999999E+09]];
    LOCAL CONST Robtarget Tr_meulage_bavure_434 := [[117.70096875,11.2087705078125,106.939],[0.607919544114108,-0.602960552027148,-0.363790158728809,0.366782116515077],[0,0,0,0],[8.999999E+09,8.999999E+09,8.999999E+09,8.999999E+09,8.999999E+09,8.999999E+09]];
    LOCAL CONST Robtarget Tr_meulage_bavure_435 := [[117.3320703125,10.49337890625,106.799765625],[0.605641405381592,-0.600424394972227,-0.367647907094864,0.370842352514397],[0,0,0,0],[8.999999E+09,8.999999E+09,8.999999E+09,8.999999E+09,8.999999E+09,8.999999E+09]];
    LOCAL CONST Robtarget Tr_meulage_bavure_436 := [[116.9165078125,9.5978828125,106.628046875],[0.603750691302616,-0.598271323556695,-0.370827533230195,0.374223819070542],[0,0,0,0],[8.999999E+09,8.999999E+09,8.999999E+09,8.999999E+09,8.999999E+09,8.999999E+09]];
    LOCAL CONST Robtarget Tr_meulage_bavure_437 := [[115.4630625,6.3165546875,106.00271875],[0.602164594889916,-0.596425841786257,-0.373481467667798,0.377075071065864],[0,0,0,0],[8.999999E+09,8.999999E+09,8.999999E+09,8.999999E+09,8.999999E+09,8.999999E+09]];
    LOCAL CONST Robtarget Tr_meulage_bavure_438 := [[115.383546875,6.13777490234375,105.9686328125],[0.600848402131503,-0.594856102616315,-0.375679146310708,0.379463560652938],[0,0,0,0],[8.999999E+09,8.999999E+09,8.999999E+09,8.999999E+09,8.999999E+09,8.999999E+09]];
    LOCAL CONST Robtarget Tr_meulage_bavure_439 := [[115.128421875,5.6400927734375,105.87184375],[0.599819820634338,-0.593586304298772,-0.377401832830904,0.381365098952421],[0,0,0,0],[8.999999E+09,8.999999E+09,8.999999E+09,8.999999E+09,8.999999E+09,8.999999E+09]];
    LOCAL CONST Robtarget Tr_meulage_bavure_440 := [[115.0727578125,5.53050048828125,105.8505625],[0.599114366011294,-0.592653432073217,-0.378603705896459,0.382731132483615],[0,0,0,0],[8.999999E+09,8.999999E+09,8.999999E+09,8.999999E+09,8.999999E+09,8.999999E+09]];
    LOCAL CONST Robtarget Tr_meulage_bavure_441 := [[113.69778125,2.82528515625,105.3251484375],[0.598746185115707,-0.592072375100733,-0.379270470802918,0.383545588462305],[0,0,0,0],[8.999999E+09,8.999999E+09,8.999999E+09,8.999999E+09,8.999999E+09,8.999999E+09]];
    LOCAL CONST Robtarget Tr_meulage_bavure_442 := [[113.61559375,2.64542114257813,105.2907265625],[0.598688435482175,-0.59181711382889,-0.379448189086118,0.383853790913174],[0,0,0,0],[8.999999E+09,8.999999E+09,8.999999E+09,8.999999E+09,8.999999E+09,8.999999E+09]];
    LOCAL CONST Robtarget Tr_meulage_bavure_443 := [[113.105078125,1.49957885742188,105.0721953125],[0.598886719821474,-0.591831192993339,-0.379223690775705,0.383744613220836],[0,0,0,0],[8.999999E+09,8.999999E+09,8.999999E+09,8.999999E+09,8.999999E+09,8.999999E+09]];
    LOCAL CONST Robtarget Tr_meulage_bavure_444 := [[112.2571640625,-0.406184234619141,104.7088046875],[0.599274574041121,-0.592043609387856,-0.378701559063442,0.383326856160315],[0,0,0,0],[8.999999E+09,8.999999E+09,8.999999E+09,8.999999E+09,8.999999E+09,8.999999E+09]];
    LOCAL CONST Robtarget Tr_meulage_bavure_445 := [[111.7022578125,-1.58114086914063,104.4829609375],[0.599789800223619,-0.592392372070184,-0.377976941886205,0.382696883268109],[0,0,0,0],[8.999999E+09,8.999999E+09,8.999999E+09,8.999999E+09,8.999999E+09,8.999999E+09]];
    LOCAL CONST Robtarget Tr_meulage_bavure_446 := [[110.30578125,-4.5777392578125,103.9080234375],[0.600386787403274,-0.5928259612191,-0.377122136654322,0.381931903958682],[0,0,0,0],[8.999999E+09,8.999999E+09,8.999999E+09,8.999999E+09,8.999999E+09,8.999999E+09]];
    LOCAL CONST Robtarget Tr_meulage_bavure_447 := [[110.255734375,-4.69199853515625,103.88628125],[0.601025177122909,-0.59330120515501,-0.376200385461213,0.381098001050678],[0,0,0,0],[8.999999E+09,8.999999E+09,8.999999E+09,8.999999E+09,8.999999E+09,8.999999E+09]];
    LOCAL CONST Robtarget Tr_meulage_bavure_448 := [[109.402796875,-6.4607109375,103.545328125],[0.601672302436405,-0.593780189485392,-0.375264700528444,0.380252457707856],[0,0,0,0],[8.999999E+09,8.999999E+09,8.999999E+09,8.999999E+09,8.999999E+09,8.999999E+09]];
    LOCAL CONST Robtarget Tr_meulage_bavure_449 := [[107.7990234375,-9.9971728515625,102.869296875],[0.60228895726808,-0.594218828802047,-0.374378892131266,0.379463358674612],[0,0,0,0],[8.999999E+09,8.999999E+09,8.999999E+09,8.999999E+09,8.999999E+09,8.999999E+09]];
    LOCAL CONST Robtarget Tr_meulage_bavure_450 := [[107.6468828125,-10.3154111328125,102.8080234375],[0.602828265538339,-0.594567353375082,-0.373618688003821,0.378809741879603],[0,0,0,0],[8.999999E+09,8.999999E+09,8.999999E+09,8.999999E+09,8.999999E+09,8.999999E+09]];
    LOCAL CONST Robtarget Tr_meulage_bavure_451 := [[107.5249921875,-10.5649150390625,102.7598359375],[0.603245722151041,-0.594780923326058,-0.373055475504983,0.378364723711952],[0,0,0,0],[8.999999E+09,8.999999E+09,8.999999E+09,8.999999E+09,8.999999E+09,8.999999E+09]];
    LOCAL CONST Robtarget Tr_meulage_bavure_452 := [[107.1634296875,-11.2775068359375,102.62146875],[0.603516640218942,-0.594829895935818,-0.372731584392414,0.378174861507405],[0,0,0,0],[8.999999E+09,8.999999E+09,8.999999E+09,8.999999E+09,8.999999E+09,8.999999E+09]];
    LOCAL CONST Robtarget Tr_meulage_bavure_453 := [[106.888796875,-11.8560576171875,102.5101875],[0.603639445158083,-0.594716219304943,-0.372648368282451,0.378239649377617],[0,0,0,0],[8.999999E+09,8.999999E+09,8.999999E+09,8.999999E+09,8.999999E+09,8.999999E+09]];
    LOCAL CONST Robtarget Tr_meulage_bavure_454 := [[106.426171875,-12.7895791015625,102.3295390625],[0.603647098986605,-0.594468308877716,-0.372755759183643,0.378511233149758],[0,0,0,0],[8.999999E+09,8.999999E+09,8.999999E+09,8.999999E+09,8.999999E+09,8.999999E+09]];
    LOCAL CONST Robtarget Tr_meulage_bavure_455 := [[104.3211171875,-17.194017578125,101.4815625],[0.603589861968556,-0.594136893075363,-0.372973750578629,0.378907920469928],[0,0,0,0],[8.999999E+09,8.999999E+09,8.999999E+09,8.999999E+09,8.999999E+09,8.999999E+09]];
    LOCAL CONST Robtarget Tr_meulage_bavure_456 := [[103.9167109375,-18.09288671875,101.3099140625],[0.603519327282365,-0.593776397673649,-0.373219348539727,0.379343286533355],[0,0,0,0],[8.999999E+09,8.999999E+09,8.999999E+09,8.999999E+09,8.999999E+09,8.999999E+09]];
    LOCAL CONST Robtarget Tr_meulage_bavure_457 := [[102.5675390625,-20.968994140625,100.7576015625],[0.603477707417064,-0.59342759988623,-0.373426741952757,0.379750982537849],[0,0,0,0],[8.999999E+09,8.999999E+09,8.999999E+09,8.999999E+09,8.999999E+09,8.999999E+09]];
    LOCAL CONST Robtarget Tr_meulage_bavure_458 := [[102.254984375,-21.63636328125,100.62946875],[0.603484612717116,-0.593113220746126,-0.373563861382905,0.380096133969452],[0,0,0,0],[8.999999E+09,8.999999E+09,8.999999E+09,8.999999E+09,8.999999E+09,8.999999E+09]];
    LOCAL CONST Robtarget Tr_meulage_bavure_459 := [[101.65296875,-22.94241015625,100.3792578125],[0.603544094958142,-0.592841318132091,-0.373622751157723,0.38036789661313],[0,0,0,0],[8.999999E+09,8.999999E+09,8.999999E+09,8.999999E+09,8.999999E+09,8.999999E+09]];
    LOCAL CONST Robtarget Tr_meulage_bavure_460 := [[100.884375,-24.602552734375,100.0610234375],[0.603653003665967,-0.592608848551093,-0.3736085081283,0.380571263284748],[0,0,0,0],[8.999999E+09,8.999999E+09,8.999999E+09,8.999999E+09,8.999999E+09,8.999999E+09]];
    LOCAL CONST Robtarget Tr_meulage_bavure_461 := [[100.8386171875,-24.6964296875,100.0428984375],[0.603808346769111,-0.592414947878446,-0.373524990393487,0.380708670053201],[0,0,0,0],[8.999999E+09,8.999999E+09,8.999999E+09,8.999999E+09,8.999999E+09,8.999999E+09]];
    LOCAL CONST Robtarget Tr_meulage_bavure_462 := [[100.799671875,-24.77847265625,100.0271171875],[0.604012475819218,-0.592263112215426,-0.373368094224568,0.380775000727135],[0,0,0,0],[8.999999E+09,8.999999E+09,8.999999E+09,8.999999E+09,8.999999E+09,8.999999E+09]];
    LOCAL CONST Robtarget Tr_meulage_bavure_463 := [[100.710703125,-24.959509765625,99.9921328125],[0.604269035481173,-0.592160976879418,-0.373130349397573,0.38075983582609],[0,0,0,0],[8.999999E+09,8.999999E+09,8.999999E+09,8.999999E+09,8.999999E+09,8.999999E+09]];
    LOCAL CONST Robtarget Tr_meulage_bavure_464 := [[99.46465625,-27.477966796875,99.5048828125],[0.604581568097142,-0.592110828636521,-0.372806775021882,0.380658643178318],[0,0,0,0],[8.999999E+09,8.999999E+09,8.999999E+09,8.999999E+09,8.999999E+09,8.999999E+09]];
    LOCAL CONST Robtarget Tr_meulage_bavure_465 := [[97.4624765625,-31.7780234375,98.67996875],[0.604943291034826,-0.592105650857728,-0.372408007998019,0.380482310276376],[0,0,0,0],[8.999999E+09,8.999999E+09,8.999999E+09,8.999999E+09,8.999999E+09,8.999999E+09]];
    LOCAL CONST Robtarget Tr_meulage_bavure_466 := [[97.3838125,-31.94680859375,98.647578125],[0.605336678422922,-0.592130824088092,-0.371960045785724,0.380255594646211],[0,0,0,0],[8.999999E+09,8.999999E+09,8.999999E+09,8.999999E+09,8.999999E+09,8.999999E+09]];
    LOCAL CONST Robtarget Tr_meulage_bavure_467 := [[97.3626171875,-31.99043359375,98.6391640625],[0.605736291652567,-0.592160194216063,-0.371502999882372,0.380020223724197],[0,0,0,0],[8.999999E+09,8.999999E+09,8.999999E+09,8.999999E+09,8.999999E+09,8.999999E+09]];
    LOCAL CONST Robtarget Tr_meulage_bavure_468 := [[97.3429296875,-32.03059765625,98.63140625],[0.606107523064234,-0.592160698827169,-0.371090464377594,0.379830547083143],[0,0,0,0],[8.999999E+09,8.999999E+09,8.999999E+09,8.999999E+09,8.999999E+09,8.999999E+09]];
    LOCAL CONST Robtarget Tr_meulage_bavure_469 := [[97.332984375,-32.0523046875,98.62725],[0.60641115810416,-0.592094796263232,-0.370783336583907,0.379748570604917],[0,0,0,0],[8.999999E+09,8.999999E+09,8.999999E+09,8.999999E+09,8.999999E+09,8.999999E+09]];
    LOCAL CONST Robtarget Tr_meulage_bavure_470 := [[96.4236328125,-33.9641171875,98.2594140625],[0.606614726274135,-0.591931863854388,-0.370631826135819,0.379825343910139],[0,0,0,0],[8.999999E+09,8.999999E+09,8.999999E+09,8.999999E+09,8.999999E+09,8.999999E+09]];
    LOCAL CONST Robtarget Tr_meulage_bavure_471 := [[96.16009375,-34.4884453125,98.1577421875],[0.606703601233569,-0.59166190937629,-0.370656609886214,0.380079732149822],[0,0,0,0],[8.999999E+09,8.999999E+09,8.999999E+09,8.999999E+09,8.999999E+09,8.999999E+09]];
    LOCAL CONST Robtarget Tr_meulage_bavure_472 := [[94.948765625,-36.85537109375,97.6975625],[0.606698570695121,-0.591305391942951,-0.370824800792011,0.380478310673889],[0,0,0,0],[8.999999E+09,8.999999E+09,8.999999E+09,8.999999E+09,8.999999E+09,8.999999E+09]];
    LOCAL CONST Robtarget Tr_meulage_bavure_473 := [[92.72065625,-41.641515625,96.7794140625],[0.606654748983795,-0.59092133598481,-0.371047877096129,0.380927109977475],[0,0,0,0],[8.999999E+09,8.999999E+09,8.999999E+09,8.999999E+09,8.999999E+09,8.999999E+09]];
    LOCAL CONST Robtarget Tr_meulage_bavure_474 := [[92.486046875,-42.14964453125,96.682046875],[0.606644426499442,-0.590587047962069,-0.37121053202845,0.381303316911573],[0,0,0,0],[8.999999E+09,8.999999E+09,8.999999E+09,8.999999E+09,8.999999E+09,8.999999E+09]];
    LOCAL CONST Robtarget Tr_meulage_bavure_475 := [[92.35884375,-42.39165234375,96.6348125],[0.606726016985809,-0.590361273390248,-0.371221838098264,0.381512062866336],[0,0,0,0],[8.999999E+09,8.999999E+09,8.999999E+09,8.999999E+09,8.999999E+09,8.999999E+09]];
    LOCAL CONST Robtarget Tr_meulage_bavure_476 := [[91.7911328125,-43.4635625,96.4253359375],[0.60690722230017,-0.590256772940126,-0.371067901520944,0.381535290607623],[0,0,0,0],[8.999999E+09,8.999999E+09,8.999999E+09,8.999999E+09,8.999999E+09,8.999999E+09]];
    LOCAL CONST Robtarget Tr_meulage_bavure_477 := [[91.136984375,-44.7838203125,96.169859375],[0.60713869797445,-0.590233617383305,-0.370821530769725,0.381442355605805],[0,0,0,0],[8.999999E+09,8.999999E+09,8.999999E+09,8.999999E+09,8.999999E+09,8.999999E+09]];
    LOCAL CONST Robtarget Tr_meulage_bavure_478 := [[89.837484375,-47.3575703125,95.670453125],[0.607342405288905,-0.590219117518981,-0.370602015795737,0.381353827752049],[0,0,0,0],[8.999999E+09,8.999999E+09,8.999999E+09,8.999999E+09,8.999999E+09,8.999999E+09]];
    LOCAL CONST Robtarget Tr_meulage_bavure_479 := [[89.5252265625,-48.020109375,95.5431484375],[0.607452484471669,-0.590154787031184,-0.370508829087347,0.381368606497308],[0,0,0,0],[8.999999E+09,8.999999E+09,8.999999E+09,8.999999E+09,8.999999E+09,8.999999E+09]];
    LOCAL CONST Robtarget Tr_meulage_bavure_480 := [[87.7587421875,-51.75019140625,94.82590625],[0.607451427922585,-0.590029573556204,-0.370566362405746,0.381508107511846],[0,0,0,0],[8.999999E+09,8.999999E+09,8.999999E+09,8.999999E+09,8.999999E+09,8.999999E+09]];
    LOCAL CONST Robtarget Tr_meulage_bavure_481 := [[87.0092578125,-53.30164453125,94.526765625],[0.607381477497619,-0.589883092991898,-0.370709798679574,0.381706592238163],[0,0,0,0],[8.999999E+09,8.999999E+09,8.999999E+09,8.999999E+09,8.999999E+09,8.999999E+09]];
    LOCAL CONST Robtarget Tr_meulage_bavure_482 := [[86.881296875,-53.55089453125,94.47828125],[0.607305555937036,-0.589782937048573,-0.370838948323875,0.381856679004583],[0,0,0,0],[8.999999E+09,8.999999E+09,8.999999E+09,8.999999E+09,8.999999E+09,8.999999E+09]];
    LOCAL CONST Robtarget Tr_meulage_bavure_483 := [[86.7188359375,-53.86798828125,94.416625],[0.607270748027289,-0.589774868389948,-0.370881170254629,0.381883491076209],[0,0,0,0],[8.999999E+09,8.999999E+09,8.999999E+09,8.999999E+09,8.999999E+09,8.999999E+09]];
    LOCAL CONST Robtarget Tr_meulage_bavure_484 := [[84.94553125,-57.44097265625,93.7250546875],[0.60727867412985,-0.589858077726459,-0.3708350629406,0.381787134646754],[0,0,0,0],[8.999999E+09,8.999999E+09,8.999999E+09,8.999999E+09,8.999999E+09,8.999999E+09]];
    LOCAL CONST Robtarget Tr_meulage_bavure_485 := [[84.8377421875,-57.72241796875,93.672359375],[0.607279394532014,-0.589984429016184,-0.370777532074295,0.381646606436075],[0,0,0,0],[8.999999E+09,8.999999E+09,8.999999E+09,8.999999E+09,8.999999E+09,8.999999E+09]];
    LOCAL CONST Robtarget Tr_meulage_bavure_486 := [[83.6523671875,-60.04382421875,93.2211796875],[0.607198384646093,-0.590077464334123,-0.370825583628282,0.381584976505798],[0,0,0,0],[8.999999E+09,8.999999E+09,8.999999E+09,8.999999E+09,8.999999E+09,8.999999E+09]];
    LOCAL CONST Robtarget Tr_meulage_bavure_487 := [[83.4616953125,-60.4566875,93.1420625],[0.606971884249142,-0.59007060352926,-0.371079908229242,0.381708679872803],[0,0,0,0],[8.999999E+09,8.999999E+09,8.999999E+09,8.999999E+09,8.999999E+09,8.999999E+09]];
    LOCAL CONST Robtarget Tr_meulage_bavure_488 := [[83.1495,-61.07697265625,93.0217578125],[0.606574855075179,-0.589935866001114,-0.371580546884822,0.382060880453386],[0,0,0,0],[8.999999E+09,8.999999E+09,8.999999E+09,8.999999E+09,8.999999E+09,8.999999E+09]];
    LOCAL CONST Robtarget Tr_meulage_bavure_489 := [[82.621328125,-62.1674453125,92.811421875],[0.606035117849179,-0.589689941510621,-0.372288394780212,0.382607579546858],[0,0,0,0],[8.999999E+09,8.999999E+09,8.999999E+09,8.999999E+09,8.999999E+09,8.999999E+09]];
    LOCAL CONST Robtarget Tr_meulage_bavure_490 := [[81.150453125,-65.20461328125,92.2256015625],[0.605419649613758,-0.589392489552722,-0.373101793457308,0.383247430310159],[0,0,0,0],[8.999999E+09,8.999999E+09,8.999999E+09,8.999999E+09,8.999999E+09,8.999999E+09]];
    LOCAL CONST Robtarget Tr_meulage_bavure_491 := [[80.1924609375,-67.276296875,91.8285390625],[0.604817337826808,-0.589124279489962,-0.373886274236318,0.383845835091655],[0,0,0,0],[8.999999E+09,8.999999E+09,8.999999E+09,8.999999E+09,8.999999E+09,8.999999E+09]];
    LOCAL CONST Robtarget Tr_meulage_bavure_492 := [[79.5739453125,-68.66740625,91.5633046875],[0.604311529448053,-0.588958284110785,-0.3745180053487,0.384281119264356],[0,0,0,0],[8.999999E+09,8.999999E+09,8.999999E+09,8.999999E+09,8.999999E+09,8.999999E+09]];
    LOCAL CONST Robtarget Tr_meulage_bavure_493 := [[78.019953125,-71.9293828125,90.9355625],[0.603955733355371,-0.58894132212718,-0.3749181274698,0.38447625275536],[0,0,0,0],[8.999999E+09,8.999999E+09,8.999999E+09,8.999999E+09,8.999999E+09,8.999999E+09]];
    LOCAL CONST Robtarget Tr_meulage_bavure_494 := [[77.3308203125,-73.3417734375,90.6628515625],[0.603769924517359,-0.589084918794303,-0.375060017823088,0.384409702957609],[0,0,0,0],[8.999999E+09,8.999999E+09,8.999999E+09,8.999999E+09,8.999999E+09,8.999999E+09]];
    LOCAL CONST Robtarget Tr_meulage_bavure_495 := [[77.1876328125,-73.64425,90.6046953125],[0.603741865246775,-0.589372357095584,-0.374964361950544,0.384106381236971],[0,0,0,0],[8.999999E+09,8.999999E+09,8.999999E+09,8.999999E+09,8.999999E+09,8.999999E+09]];
    LOCAL CONST Robtarget Tr_meulage_bavure_496 := [[76.7251953125,-74.656078125,90.4110703125],[0.603839665006292,-0.58976946358096,-0.374680757937615,0.383619562097412],[0,0,0,0],[8.999999E+09,8.999999E+09,8.999999E+09,8.999999E+09,8.999999E+09,8.999999E+09]];
    LOCAL CONST Robtarget Tr_meulage_bavure_497 := [[76.29028125,-75.6409375,90.2234609375],[0.604022344998859,-0.590230780114226,-0.37427381682012,0.383019246240617],[0,0,0,0],[8.999999E+09,8.999999E+09,8.999999E+09,8.999999E+09,8.999999E+09,8.999999E+09]];
    LOCAL CONST Robtarget Tr_meulage_bavure_498 := [[75.7788671875,-76.7015625,90.0190078125],[0.604241184890217,-0.59070542862663,-0.373819543519731,0.382385454687016],[0,0,0,0],[8.999999E+09,8.999999E+09,8.999999E+09,8.999999E+09,8.999999E+09,8.999999E+09]];
    LOCAL CONST Robtarget Tr_meulage_bavure_499 := [[75.463265625,-77.3057421875,89.9011796875],[0.604443479835091,-0.591139416066408,-0.373400439986691,0.381804114534218],[0,0,0,0],[8.999999E+09,8.999999E+09,8.999999E+09,8.999999E+09,8.999999E+09,8.999999E+09]];
    LOCAL CONST Robtarget Tr_meulage_bavure_500 := [[74.9770703125,-78.3100390625,89.707484375],[0.604577995229211,-0.591483379049179,-0.373095980259887,0.381355804344326],[0,0,0,0],[8.999999E+09,8.999999E+09,8.999999E+09,8.999999E+09,8.999999E+09,8.999999E+09]];
    LOCAL CONST Robtarget Tr_meulage_bavure_501 := [[74.218890625,-79.88609375,89.4037734375],[0.604606276771825,-0.59169958032628,-0.372966579109235,0.381102069788883],[0,0,0,0],[8.999999E+09,8.999999E+09,8.999999E+09,8.999999E+09,8.999999E+09,8.999999E+09]];
    LOCAL CONST Robtarget Tr_meulage_bavure_502 := [[73.417234375,-81.605203125,89.07390625],[0.604513886231304,-0.591774711961752,-0.37303482925314,0.381065175265586],[0,0,0,0],[8.999999E+09,8.999999E+09,8.999999E+09,8.999999E+09,8.999999E+09,8.999999E+09]];
    LOCAL CONST Robtarget Tr_meulage_bavure_503 := [[73.01615625,-82.461859375,88.9094453125],[0.604313024922432,-0.591720535552931,-0.37328197510488,0.381225842219349],[0,0,0,0],[8.999999E+09,8.999999E+09,8.999999E+09,8.999999E+09,8.999999E+09,8.999999E+09]];
    LOCAL CONST Robtarget Tr_meulage_bavure_504 := [[72.920390625,-82.664015625,88.8705703125],[0.604034226190077,-0.591574708480491,-0.373656836512698,0.381526652285918],[0,0,0,0],[8.999999E+09,8.999999E+09,8.999999E+09,8.999999E+09,8.999999E+09,8.999999E+09]];
    LOCAL CONST Robtarget Tr_meulage_bavure_505 := [[72.4820390625,-83.599390625,88.6909765625],[0.603724467917129,-0.591387258530817,-0.374084416910778,0.38188836891179],[0,0,0,0],[8.999999E+09,8.999999E+09,8.999999E+09,8.999999E+09,8.999999E+09,8.999999E+09]];
    LOCAL CONST Robtarget Tr_meulage_bavure_506 := [[71.4756171875,-85.72271875,88.282640625],[0.603436651073866,-0.591207758156231,-0.374483684557306,0.382229727830037],[0,0,0,0],[8.999999E+09,8.999999E+09,8.999999E+09,8.999999E+09,8.999999E+09,8.999999E+09]];
    LOCAL CONST Robtarget Tr_meulage_bavure_507 := [[69.368953125,-90.0317265625,87.4503984375],[0.603211839059123,-0.591082528598805,-0.374788532660905,0.382479381653494],[0,0,0,0],[8.999999E+09,8.999999E+09,8.999999E+09,8.999999E+09,8.999999E+09,8.999999E+09]];
    LOCAL CONST Robtarget Tr_meulage_bavure_508 := [[69.2497265625,-90.2794375,87.40265625],[0.603074580196487,-0.591039342054224,-0.37495962125375,0.382594863130944],[0,0,0,0],[8.999999E+09,8.999999E+09,8.999999E+09,8.999999E+09,8.999999E+09,8.999999E+09]];
    LOCAL CONST Robtarget Tr_meulage_bavure_509 := [[69.213453125,-90.35771875,87.3876484375],[0.603031491675562,-0.591073893771276,-0.37499173510666,0.382577927684421],[0,0,0,0],[8.999999E+09,8.999999E+09,8.999999E+09,8.999999E+09,8.999999E+09,8.999999E+09]];
    LOCAL CONST Robtarget Tr_meulage_bavure_510 := [[68.8040078125,-91.30140625,87.2082890625],[0.603058387176764,-0.591162912965547,-0.374922039899278,0.382466280850501],[0,0,0,0],[8.999999E+09,8.999999E+09,8.999999E+09,8.999999E+09,8.999999E+09,8.999999E+09]];
    LOCAL CONST Robtarget Tr_meulage_bavure_511 := [[68.4482109375,-92.1153671875,87.0534375],[0.603098630714043,-0.591279739342971,-0.374825033194103,0.382317284417529],[0,0,0,0],[8.999999E+09,8.999999E+09,8.999999E+09,8.999999E+09,8.999999E+09,8.999999E+09]];
    LOCAL CONST Robtarget Tr_meulage_bavure_512 := [[67.1682734375,-94.7817109375,86.5397734375],[0.603131251477706,-0.591352533412559,-0.374756204000515,0.382220698393755],[0,0,0,0],[8.999999E+09,8.999999E+09,8.999999E+09,8.999999E+09,8.999999E+09,8.999999E+09]];
    LOCAL CONST Robtarget Tr_meulage_bavure_513 := [[67.1298359375,-94.868375,86.5232578125],[0.603141520995614,-0.591344207911111,-0.374748598645459,0.382224830740158],[0,0,0,0],[8.999999E+09,8.999999E+09,8.999999E+09,8.999999E+09,8.999999E+09,8.999999E+09]];
    LOCAL CONST Robtarget Tr_meulage_bavure_514 := [[67.03265625,-95.05571875,86.4867578125],[0.60313413910232,-0.59126879138267,-0.374790704063037,0.382311855340785],[0,0,0,0],[8.999999E+09,8.999999E+09,8.999999E+09,8.999999E+09,8.999999E+09,8.999999E+09]];
    LOCAL CONST Robtarget Tr_meulage_bavure_515 := [[66.21346875,-96.585421875,86.1873203125],[0.603177369264715,-0.591171461795596,-0.374786681103913,0.382398100979163],[0,0,0,0],[8.999999E+09,8.999999E+09,8.999999E+09,8.999999E+09,8.999999E+09,8.999999E+09]];
    LOCAL CONST Robtarget Tr_meulage_bavure_516 := [[65.6870859375,-97.7146796875,85.97065625],[0.603397432678364,-0.591132002851046,-0.374561124971763,0.382332913966818],[0,0,0,0],[8.999999E+09,8.999999E+09,8.999999E+09,8.999999E+09,8.999999E+09,8.999999E+09]];
    LOCAL CONST Robtarget Tr_meulage_bavure_517 := [[64.5423046875,-100.056625,85.51834375],[0.603922110604293,-0.591257170758994,-0.373924406199566,0.381934000578147],[0,0,0,0],[8.999999E+09,8.999999E+09,8.999999E+09,8.999999E+09,8.999999E+09,8.999999E+09]];
    LOCAL CONST Robtarget Tr_meulage_bavure_518 := [[64.46765234375,-100.211796875,85.4884375],[0.604847453242577,-0.591568505771905,-0.372758811137628,0.38112613398195],[0,0,0,0],[8.999999E+09,8.999999E+09,8.999999E+09,8.999999E+09,8.999999E+09,8.999999E+09]];
    LOCAL CONST Robtarget Tr_meulage_bavure_519 := [[64.3466328125,-100.4663515625,85.43946875],[0.606107336895317,-0.592009424566849,-0.371159997309558,0.379998676027778],[0,0,0,0],[8.999999E+09,8.999999E+09,8.999999E+09,8.999999E+09,8.999999E+09,8.999999E+09]];
    LOCAL CONST Robtarget Tr_meulage_bavure_520 := [[63.359328125,-102.5683984375,85.035734375],[0.607477577432725,-0.59233245034933,-0.369487945253474,0.378935244457403],[0,0,0,0],[8.999999E+09,8.999999E+09,8.999999E+09,8.999999E+09,8.999999E+09,8.999999E+09]];
    LOCAL CONST Robtarget Tr_meulage_bavure_521 := [[63.097734375,-103.0585390625,84.9398359375],[0.608570455879613,-0.592126665989224,-0.368365820040457,0.378595607846799],[0,0,0,0],[8.999999E+09,8.999999E+09,8.999999E+09,8.999999E+09,8.999999E+09,8.999999E+09]];
    LOCAL CONST Robtarget Tr_meulage_bavure_522 := [[61.8127109375,-105.398421875,84.4800234375],[0.608910085373308,-0.590945599293452,-0.368530118893265,0.37973327227791],[0,0,0,0],[8.999999E+09,8.999999E+09,8.999999E+09,8.999999E+09,8.999999E+09,8.999999E+09]];
    LOCAL CONST Robtarget Tr_meulage_bavure_523 := [[61.7417734375,-105.5559921875,84.4499296875],[0.60813563878345,-0.588416230625268,-0.370527487875233,0.382944859094707],[0,0,0,0],[8.999999E+09,8.999999E+09,8.999999E+09,8.999999E+09,8.999999E+09,8.999999E+09]];
    LOCAL CONST Robtarget Tr_meulage_bavure_524 := [[61.65121484375,-105.766828125,84.40990625],[0.606121600473602,-0.584431976939605,-0.374469236914731,0.388366657135088],[0,0,0,0],[8.999999E+09,8.999999E+09,8.999999E+09,8.999999E+09,8.999999E+09,8.999999E+09]];
    LOCAL CONST Robtarget Tr_meulage_bavure_525 := [[60.93575,-107.698890625,84.0495546875],[0.603046552654832,-0.57926748340493,-0.379927627992275,0.395523748324933],[0,0,0,0],[8.999999E+09,8.999999E+09,8.999999E+09,8.999999E+09,8.999999E+09,8.999999E+09]];
    LOCAL CONST Robtarget Tr_meulage_bavure_526 := [[60.6432734375,-108.4778359375,83.9040546875],[0.599506401041337,-0.573532275284584,-0.385913177618239,0.403390410964297],[0,0,0,0],[8.999999E+09,8.999999E+09,8.999999E+09,8.999999E+09,8.999999E+09,8.999999E+09]];
    LOCAL CONST Robtarget Tr_meulage_bavure_527 := [[60.58623828125,-108.6301328125,83.875609375],[0.596345875866182,-0.568102057592842,-0.391176684551428,0.410624463420689],[0,0,0,0],[8.999999E+09,8.999999E+09,8.999999E+09,8.999999E+09,8.999999E+09,8.999999E+09]];
    LOCAL CONST Robtarget Tr_meulage_bavure_528 := [[60.5231328125,-108.83778125,83.83765625],[0.594507807382365,-0.563926765218748,-0.394469764377703,0.415861365629379],[0,0,0,0],[8.999999E+09,8.999999E+09,8.999999E+09,8.999999E+09,8.999999E+09,8.999999E+09]];
    LOCAL CONST Robtarget Tr_meulage_bavure_529 := [[60.326328125,-109.2331953125,83.7610859375],[0.594823937460528,-0.561890835988626,-0.394753734587202,0.417890728403267],[0,0,0,0],[8.999999E+09,8.999999E+09,8.999999E+09,8.999999E+09,8.999999E+09,8.999999E+09]];
    LOCAL CONST Robtarget Tr_meulage_bavure_530 := [[59.554046875,-111.0446796875,83.4175546875],[0.597934739912994,-0.562720620670476,-0.39119502435754,0.415675357454971],[0,0,0,0],[8.999999E+09,8.999999E+09,8.999999E+09,8.999999E+09,8.999999E+09,8.999999E+09]];
    LOCAL CONST Robtarget Tr_meulage_bavure_531 := [[59.051203125,-111.83971875,83.2576171875],[0.604226013845415,-0.566857425764697,-0.383139270762454,0.40839672164149],[0,0,0,0],[8.999999E+09,8.999999E+09,8.999999E+09,8.999999E+09,8.999999E+09,8.999999E+09]];
    LOCAL CONST Robtarget Tr_meulage_bavure_532 := [[58.8616484375,-112.109796875,83.202234375],[0.613785253299694,-0.574486496491518,-0.37003946101198,0.395352659627699],[0,0,0,0],[8.999999E+09,8.999999E+09,8.999999E+09,8.999999E+09,8.999999E+09,8.999999E+09]];
    LOCAL CONST Robtarget Tr_meulage_bavure_533 := [[58.77103515625,-112.19634375,83.1828203125],[0.626428103313937,-0.585595377806249,-0.351321125158034,0.375818243155056],[0,0,0,0],[8.999999E+09,8.999999E+09,8.999999E+09,8.999999E+09,8.999999E+09,8.999999E+09]];
    LOCAL CONST Robtarget Tr_meulage_bavure_534 := [[57.6429765625,-113.370171875,82.925125],[0.641731009859323,-0.599946522356388,-0.326267671812212,0.348991242909688],[0,0,0,0],[8.999999E+09,8.999999E+09,8.999999E+09,8.999999E+09,8.999999E+09,8.999999E+09]];
    LOCAL CONST Robtarget Tr_meulage_bavure_535 := [[56.38540625,-114.1503359375,82.725453125],[0.659006477795059,-0.617089707254816,-0.293918422357325,0.313883284714712],[0,0,0,0],[8.999999E+09,8.999999E+09,8.999999E+09,8.999999E+09,8.999999E+09,8.999999E+09]];
    LOCAL CONST Robtarget Tr_meulage_bavure_536 := [[56.2052734375,-114.233109375,82.7016640625],[0.677211248151706,-0.636162598033539,-0.253127035632003,0.269460160454533],[0,0,0,0],[8.999999E+09,8.999999E+09,8.999999E+09,8.999999E+09,8.999999E+09,8.999999E+09]];
    LOCAL CONST Robtarget Tr_meulage_bavure_537 := [[56.11117578125,-114.2425625,82.6948359375],[0.694612613587334,-0.655739000229462,-0.203082323294063,0.215121478678735],[0,0,0,0],[8.999999E+09,8.999999E+09,8.999999E+09,8.999999E+09,8.999999E+09,8.999999E+09]];
    LOCAL CONST Robtarget Tr_meulage_bavure_538 := [[53.22722265625,-114.68078125,82.4609375],[0.708730380786893,-0.673528844580681,-0.144598525810513,0.152155871398069],[0,0,0,0],[8.999999E+09,8.999999E+09,8.999999E+09,8.999999E+09,8.999999E+09,8.999999E+09]];
    LOCAL CONST Robtarget Tr_meulage_bavure_539 := [[52.94658203125,-114.6301796875,82.4536328125],[0.717020579109376,-0.68702192649238,-0.0815150710623826,0.0850744076796795],[0,0,0,0],[8.999999E+09,8.999999E+09,8.999999E+09,8.999999E+09,8.999999E+09,8.999999E+09]];
    LOCAL CONST Robtarget Tr_meulage_bavure_540 := [[51.30771484375,-114.32615625,82.4124140625],[0.718391382543388,-0.695006582688426,-0.0206224511212573,0.0213163321635403],[0,0,0,0],[8.999999E+09,8.999999E+09,8.999999E+09,8.999999E+09,8.999999E+09,8.999999E+09]];
    LOCAL CONST Robtarget Tr_meulage_bavure_541 := [[48.41323046875,-113.292015625,82.4220625],[0.714253629371172,-0.698494765163511,0.0308495450293432,-0.0315455470829474],[0,0,0,0],[8.999999E+09,8.999999E+09,8.999999E+09,8.999999E+09,8.999999E+09,8.999999E+09]];
    LOCAL CONST Robtarget Tr_meulage_bavure_542 := [[47.8818203125,-113.07315625,82.428640625],[0.707554547223755,-0.700000218320891,0.0680651260908972,-0.0687996777893795],[0,0,0,0],[8.999999E+09,8.999999E+09,8.999999E+09,8.999999E+09,8.999999E+09,8.999999E+09]];
    LOCAL CONST Robtarget Tr_meulage_bavure_543 := [[47.335375,-112.759875,82.45003125],[0.700994974833916,-0.701898444864228,0.0893452717447061,-0.0892302682481717],[0,0,0,0],[8.999999E+09,8.999999E+09,8.999999E+09,8.999999E+09,8.999999E+09,8.999999E+09]];
    LOCAL CONST Robtarget Tr_meulage_bavure_544 := [[43.7784453125,-110.9981484375,82.5432734375],[0.696095825867166,-0.705386739472806,0.0951766935123562,-0.0939230855449671],[0,0,0,0],[8.999999E+09,8.999999E+09,8.999999E+09,8.999999E+09,8.999999E+09,8.999999E+09]];
    LOCAL CONST Robtarget Tr_meulage_bavure_545 := [[42.5384921875,-110.4135703125,82.570875],[0.693104650242598,-0.71047331708963,0.0871799066269696,-0.0850486531125351],[0,0,0,0],[8.999999E+09,8.999999E+09,8.999999E+09,8.999999E+09,8.999999E+09,8.999999E+09]];
    LOCAL CONST Robtarget Tr_meulage_bavure_546 := [[40.288171875,-109.8341328125,82.541140625],[0.691401433678135,-0.716272027232614,0.0679466036277191,-0.0655873430423779],[0,0,0,0],[8.999999E+09,8.999999E+09,8.999999E+09,8.999999E+09,8.999999E+09,8.999999E+09]];
    LOCAL CONST Robtarget Tr_meulage_bavure_547 := [[40.21958984375,-109.8151796875,82.5404453125],[0.690064923269362,-0.721538975078166,0.0408299902802154,-0.039048956581664],[0,0,0,0],[8.999999E+09,8.999999E+09,8.999999E+09,8.999999E+09,8.999999E+09,8.999999E+09]];
    LOCAL CONST Robtarget Tr_meulage_bavure_548 := [[40.04356640625,-109.8084453125,82.5317265625],[0.688340392068972,-0.725272732667709,0.00937247079318892,-0.00889520580307608],[0,0,0,0],[8.999999E+09,8.999999E+09,8.999999E+09,8.999999E+09,8.999999E+09,8.999999E+09]];
    LOCAL CONST Robtarget Tr_meulage_bavure_549 := [[36.89140625,-109.8212265625,82.3533671875],[0.685948248195779,-0.726909195914964,-0.0238796594244099,0.0225340532789216],[0,0,0,0],[8.999999E+09,8.999999E+09,8.999999E+09,8.999999E+09,8.999999E+09,8.999999E+09]];
    LOCAL CONST Robtarget Tr_meulage_bavure_550 := [[36.6884921875,-109.8885234375,82.3308671875],[0.682834643678899,-0.726280488692536,-0.057614021173935,0.0541675705622144],[0,0,0,0],[8.999999E+09,8.999999E+09,8.999999E+09,8.999999E+09,8.999999E+09,8.999999E+09]];
    LOCAL CONST Robtarget Tr_meulage_bavure_551 := [[36.48870703125,-109.9717578125,82.3058984375],[0.679030252672373,-0.723374402186131,-0.0912029202917883,0.0856120175431038],[0,0,0,0],[8.999999E+09,8.999999E+09,8.999999E+09,8.999999E+09,8.999999E+09,8.999999E+09]];
    LOCAL CONST Robtarget Tr_meulage_bavure_552 := [[35.92006640625,-110.274328125,82.2239375],[0.674578626234751,-0.718307008918738,-0.124089579795307,0.11653537725376],[0,0,0,0],[8.999999E+09,8.999999E+09,8.999999E+09,8.999999E+09,8.999999E+09,8.999999E+09]];
    LOCAL CONST Robtarget Tr_meulage_bavure_553 := [[34.6355,-110.747453125,82.073671875],[0.669628141379067,-0.71136137716403,-0.15542594618335,0.146307616361972],[0,0,0,0],[8.999999E+09,8.999999E+09,8.999999E+09,8.999999E+09,8.999999E+09,8.999999E+09]];
    LOCAL CONST Robtarget Tr_meulage_bavure_554 := [[33.56742578125,-111.23784375,81.9326484375],[0.664389458163375,-0.702972985711214,-0.184455998778801,0.174331906879244],[0,0,0,0],[8.999999E+09,8.999999E+09,8.999999E+09,8.999999E+09,8.999999E+09,8.999999E+09]];
    LOCAL CONST Robtarget Tr_meulage_bavure_555 := [[32.282806640625,-112.1738984375,81.7056171875],[0.659068586085261,-0.693594707835663,-0.210794479725018,0.200301441371238],[0,0,0,0],[8.999999E+09,8.999999E+09,8.999999E+09,8.999999E+09,8.999999E+09,8.999999E+09]];
    LOCAL CONST Robtarget Tr_meulage_bavure_556 := [[32.260259765625,-112.1936640625,81.701078125],[0.653766680242046,-0.683600560835054,-0.234493276534986,0.224259457528954],[0,0,0,0],[8.999999E+09,8.999999E+09,8.999999E+09,8.999999E+09,8.999999E+09,8.999999E+09]];
    LOCAL CONST Robtarget Tr_meulage_bavure_557 := [[30.800005859375,-113.795109375,81.35390625],[0.648499742433259,-0.673288508782455,-0.255792791274249,0.246375152841399],[0,0,0,0],[8.999999E+09,8.999999E+09,8.999999E+09,8.999999E+09,8.999999E+09,8.999999E+09]];
    LOCAL CONST Robtarget Tr_meulage_bavure_558 := [[30.36337109375,-114.3786328125,81.2327421875],[0.643227527681142,-0.66283982458125,-0.275056866760639,0.26691840444249],[0,0,0,0],[8.999999E+09,8.999999E+09,8.999999E+09,8.999999E+09,8.999999E+09,8.999999E+09]];
    LOCAL CONST Robtarget Tr_meulage_bavure_559 := [[29.2110078125,-116.3321328125,80.8444140625],[0.637851784835453,-0.652366742623963,-0.292687903696435,0.286175688572971],[0,0,0,0],[8.999999E+09,8.999999E+09,8.999999E+09,8.999999E+09,8.999999E+09,8.999999E+09]];
    LOCAL CONST Robtarget Tr_meulage_bavure_560 := [[29.06588671875,-116.5931796875,80.793015625],[0.632267838338525,-0.641983684711661,-0.309000409408019,0.304323965787193],[0,0,0,0],[8.999999E+09,8.999999E+09,8.999999E+09,8.999999E+09,8.999999E+09,8.999999E+09]];
    LOCAL CONST Robtarget Tr_meulage_bavure_561 := [[28.67373828125,-117.407671875,80.6360390625],[0.626516445166425,-0.631834540546292,-0.324054439200274,0.321326901680014],[0,0,0,0],[8.999999E+09,8.999999E+09,8.999999E+09,8.999999E+09,8.999999E+09,8.999999E+09]];
    LOCAL CONST Robtarget Tr_meulage_bavure_562 := [[26.621146484375,-121.66309375,79.815703125],[0.620805329766407,-0.622234038428185,-0.337600602916891,0.336825439753482],[0,0,0,0],[8.999999E+09,8.999999E+09,8.999999E+09,8.999999E+09,8.999999E+09,8.999999E+09]];
    LOCAL CONST Robtarget Tr_meulage_bavure_563 := [[26.25398046875,-122.401578125,79.6727265625],[0.615533340640601,-0.613640896064988,-0.349149320323023,0.350226083201054],[0,0,0,0],[8.999999E+09,8.999999E+09,8.999999E+09,8.999999E+09,8.999999E+09,8.999999E+09]];
    LOCAL CONST Robtarget Tr_meulage_bavure_564 := [[24.520607421875,-126.0058671875,78.978203125],[0.611189645186933,-0.606487847916517,-0.358205618336633,0.360982607528302],[0,0,0,0],[8.999999E+09,8.999999E+09,8.999999E+09,8.999999E+09,8.999999E+09,8.999999E+09]];
    LOCAL CONST Robtarget Tr_meulage_bavure_565 := [[24.40336328125,-126.26328125,78.92896875],[0.608071435187378,-0.601079492600946,-0.364583480571098,0.368824428391634],[0,0,0,0],[8.999999E+09,8.999999E+09,8.999999E+09,8.999999E+09,8.999999E+09,8.999999E+09]];
    LOCAL CONST Robtarget Tr_meulage_bavure_566 := [[23.8350234375,-127.547875,78.6841953125],[0.606216536350926,-0.597392538498787,-0.3684986658179,0.373941705739129],[0,0,0,0],[8.999999E+09,8.999999E+09,8.999999E+09,8.999999E+09,8.999999E+09,8.999999E+09]];
    LOCAL CONST Robtarget Tr_meulage_bavure_567 := [[22.022978515625,-131.29403125,77.96175],[0.605368788802514,-0.595083226915675,-0.370551626421752,0.376956330021926],[0,0,0,0],[8.999999E+09,8.999999E+09,8.999999E+09,8.999999E+09,8.999999E+09,8.999999E+09]];
    LOCAL CONST Robtarget Tr_meulage_bavure_568 := [[21.647296875,-132.05375,77.8147734375],[0.605116978552125,-0.593657573437963,-0.371500057460674,0.37867114370442],[0,0,0,0],[8.999999E+09,8.999999E+09,8.999999E+09,8.999999E+09,8.999999E+09,8.999999E+09]];
    LOCAL CONST Robtarget Tr_meulage_bavure_569 := [[21.279955078125,-132.89521875,77.65471875],[0.605037801425412,-0.592626498410401,-0.372064541522466,0.379856642919151],[0,0,0,0],[8.999999E+09,8.999999E+09,8.999999E+09,8.999999E+09,8.999999E+09,8.999999E+09]];
    LOCAL CONST Robtarget Tr_meulage_bavure_570 := [[21.0843984375,-133.3335,77.571109375],[0.604823625443045,-0.591655602992695,-0.372745674688986,0.38104158769606],[0,0,0,0],[8.999999E+09,8.999999E+09,8.999999E+09,8.999999E+09,8.999999E+09,8.999999E+09]];
    LOCAL CONST Robtarget Tr_meulage_bavure_571 := [[20.079779296875,-135.3951875,77.1731015625],[0.604377891805029,-0.590569702306456,-0.373729169927206,0.382467381825555],[0,0,0,0],[8.999999E+09,8.999999E+09,8.999999E+09,8.999999E+09,8.999999E+09,8.999999E+09]];
    LOCAL CONST Robtarget Tr_meulage_bavure_572 := [[19.30170703125,-137.03159375,76.8582734375],[0.603769893422824,-0.589337997832733,-0.37494858509356,0.384130444827061],[0,0,0,0],[8.999999E+09,8.999999E+09,8.999999E+09,8.999999E+09,8.999999E+09,8.999999E+09]];
    LOCAL CONST Robtarget Tr_meulage_bavure_573 := [[18.45233984375,-138.92234375,76.4972890625],[0.603156278273041,-0.588087282296953,-0.376172260532503,0.385811200960088],[0,0,0,0],[8.999999E+09,8.999999E+09,8.999999E+09,8.999999E+09,8.999999E+09,8.999999E+09]];
    LOCAL CONST Robtarget Tr_meulage_bavure_574 := [[17.20995703125,-141.27996875,76.0369140625],[0.602735031664773,-0.586994027180106,-0.377106855503652,0.387219463858796],[0,0,0,0],[8.999999E+09,8.999999E+09,8.999999E+09,8.999999E+09,8.999999E+09,8.999999E+09]];
    LOCAL CONST Robtarget Tr_meulage_bavure_575 := [[16.98721484375,-141.711203125,75.9529609375],[0.602702042414475,-0.586226331539901,-0.377470176957368,0.388078860267425],[0,0,0,0],[8.999999E+09,8.999999E+09,8.999999E+09,8.999999E+09,8.999999E+09,8.999999E+09]];
    LOCAL CONST Robtarget Tr_meulage_bavure_576 := [[16.178705078125,-143.628140625,75.5899140625],[0.603246885757168,-0.585906830296111,-0.377007215909961,0.388164836362676],[0,0,0,0],[8.999999E+09,8.999999E+09,8.999999E+09,8.999999E+09,8.999999E+09,8.999999E+09]];
    LOCAL CONST Robtarget Tr_meulage_bavure_577 := [[15.4666005859375,-145.2381875,75.283140625],[0.604477026196554,-0.586115994009111,-0.375566179074331,0.387331397517409],[0,0,0,0],[8.999999E+09,8.999999E+09,8.999999E+09,8.999999E+09,8.999999E+09,8.999999E+09]];
    LOCAL CONST Robtarget Tr_meulage_bavure_578 := [[15.2182099609375,-145.7295625,75.18778125],[0.606435727306895,-0.586895519168113,-0.373073094820273,0.385494259551776],[0,0,0,0],[8.999999E+09,8.999999E+09,8.999999E+09,8.999999E+09,8.999999E+09,8.999999E+09]];
    LOCAL CONST Robtarget Tr_meulage_bavure_579 := [[13.9345048828125,-148.106375,74.721921875],[0.609185398333783,-0.588283778406105,-0.36942209360887,0.382547596090717],[0,0,0,0],[8.999999E+09,8.999999E+09,8.999999E+09,8.999999E+09,8.999999E+09,8.999999E+09]];
    LOCAL CONST Robtarget Tr_meulage_bavure_580 := [[13.7811552734375,-148.393921875,74.6656640625],[0.612832833193754,-0.590369478093531,-0.364418363366499,0.378284356452353],[0,0,0,0],[8.999999E+09,8.999999E+09,8.999999E+09,8.999999E+09,8.999999E+09,8.999999E+09]];
    LOCAL CONST Robtarget Tr_meulage_bavure_581 := [[13.7513310546875,-148.450578125,74.654609375],[0.61759381517864,-0.593330952753912,-0.357672730759229,0.372298908981027],[0,0,0,0],[8.999999E+09,8.999999E+09,8.999999E+09,8.999999E+09,8.999999E+09,8.999999E+09]];
    LOCAL CONST Robtarget Tr_meulage_bavure_582 := [[13.7377197265625,-148.47125,74.6504140625],[0.623793541581112,-0.597417056861548,-0.348574660600993,0.363964536238741],[0,0,0,0],[8.999999E+09,8.999999E+09,8.999999E+09,8.999999E+09,8.999999E+09,8.999999E+09]];
    LOCAL CONST Robtarget Tr_meulage_bavure_583 := [[12.59455859375,-149.8640625,74.3555703125],[0.631769520032377,-0.602951630989445,-0.336336802578706,0.35241191733022],[0,0,0,0],[8.999999E+09,8.999999E+09,8.999999E+09,8.999999E+09,8.999999E+09,8.999999E+09]];
    LOCAL CONST Robtarget Tr_meulage_bavure_584 := [[12.1518154296875,-150.409828125,74.2403203125],[0.641786298316294,-0.610137406017366,-0.320106674781439,0.336711166776866],[0,0,0,0],[8.999999E+09,8.999999E+09,8.999999E+09,8.999999E+09,8.999999E+09,8.999999E+09]];
    LOCAL CONST Robtarget Tr_meulage_bavure_585 := [[12.1244296875,-150.433703125,74.234828125],[0.653925432932289,-0.618992260049319,-0.299041549171371,0.315918125520746],[0,0,0,0],[8.999999E+09,8.999999E+09,8.999999E+09,8.999999E+09,8.999999E+09,8.999999E+09]];
    LOCAL CONST Robtarget Tr_meulage_bavure_586 := [[12.1081708984375,-150.444859375,74.2320703125],[0.668049420189305,-0.629348873792321,-0.272244677451326,0.28898581771515],[0,0,0,0],[8.999999E+09,8.999999E+09,8.999999E+09,8.999999E+09,8.999999E+09,8.999999E+09]];
    LOCAL CONST Robtarget Tr_meulage_bavure_587 := [[10.8476552734375,-151.255671875,74.02715625],[0.683762862214142,-0.640754506124172,-0.238740232872013,0.254764817717261],[0,0,0,0],[8.999999E+09,8.999999E+09,8.999999E+09,8.999999E+09,8.999999E+09,8.999999E+09]];
    LOCAL CONST Robtarget Tr_meulage_bavure_588 := [[8.8689619140625,-151.6510625,73.8509765625],[0.700245963739753,-0.652389764184977,-0.197615448799607,0.212111574999066],[0,0,0,0],[8.999999E+09,8.999999E+09,8.999999E+09,8.999999E+09,8.999999E+09,8.999999E+09]];
    LOCAL CONST Robtarget Tr_meulage_bavure_589 := [[8.8024013671875,-151.65940625,73.8458671875],[0.715998296646655,-0.662885557944203,-0.148731826611834,0.160648747336539],[0,0,0,0],[8.999999E+09,8.999999E+09,8.999999E+09,8.999999E+09,8.999999E+09,8.999999E+09]];
    LOCAL CONST Robtarget Tr_meulage_bavure_590 := [[8.5939326171875,-151.630578125,73.8389921875],[0.728979192958908,-0.670325696516845,-0.0939191693312916,0.102137096367117],[0,0,0,0],[8.999999E+09,8.999999E+09,8.999999E+09,8.999999E+09,8.999999E+09,8.999999E+09]];
    LOCAL CONST Robtarget Tr_meulage_bavure_591 := [[6.363822265625,-150.999515625,73.8189453125],[0.737384893686962,-0.673143622087706,-0.0377865724675259,0.0413927233468327],[0,0,0,0],[8.999999E+09,8.999999E+09,8.999999E+09,8.999999E+09,8.999999E+09,8.999999E+09]];
    LOCAL CONST Robtarget Tr_meulage_bavure_592 := [[5.11608056640625,-150.663734375,73.804859375],[0.740963792674772,-0.671237226005034,0.0136480077410071,-0.0150657311401192],[0,0,0,0],[8.999999E+09,8.999999E+09,8.999999E+09,8.999999E+09,8.999999E+09,8.999999E+09]];
    LOCAL CONST Robtarget Tr_meulage_bavure_593 := [[5.07372607421875,-150.647140625,73.80525],[0.741180368325717,-0.666083760098068,0.05586059208503,-0.0621585102305743],[0,0,0,0],[8.999999E+09,8.999999E+09,8.999999E+09,8.999999E+09,8.999999E+09,8.999999E+09]];
    LOCAL CONST Robtarget Tr_meulage_bavure_594 := [[4.05832958984375,-150.213609375,73.820359375],[0.740035949740323,-0.659613290113963,0.0874084372028521,-0.0980656193715476],[0,0,0,0],[8.999999E+09,8.999999E+09,8.999999E+09,8.999999E+09,8.999999E+09,8.999999E+09]];
    LOCAL CONST Robtarget Tr_meulage_bavure_595 := [[2.39737719726563,-149.451703125,73.853828125],[0.738983788537122,-0.653219214884323,0.109243128294232,-0.123586231052334],[0,0,0,0],[8.999999E+09,8.999999E+09,8.999999E+09,8.999999E+09,8.999999E+09,8.999999E+09]];
    LOCAL CONST Robtarget Tr_meulage_bavure_596 := [[-1.05331433105469,-148.01134375,73.8997265625],[0.738667891967023,-0.647553679621989,0.123403850430462,-0.140767421955342],[0,0,0,0],[8.999999E+09,8.999999E+09,8.999999E+09,8.999999E+09,8.999999E+09,8.999999E+09]];
    LOCAL CONST Robtarget Tr_meulage_bavure_597 := [[-2.98388549804688,-147.14828125,73.934890625],[0.739173484405913,-0.642786374601908,0.131972138619869,-0.151761626261235],[0,0,0,0],[8.999999E+09,8.999999E+09,8.999999E+09,8.999999E+09,8.999999E+09,8.999999E+09]];
    LOCAL CONST Robtarget Tr_meulage_bavure_598 := [[-3.14477001953125,-147.075484375,73.93796875],[0.740362878518013,-0.6388443146203,0.136631337959784,-0.158343384065015],[0,0,0,0],[8.999999E+09,8.999999E+09,8.999999E+09,8.999999E+09,8.999999E+09,8.999999E+09]];
    LOCAL CONST Robtarget Tr_meulage_bavure_599 := [[-3.39498657226562,-146.960359375,73.9430703125],[0.742030256064681,-0.635637695321563,0.138549635672086,-0.161739969784858],[0,0,0,0],[8.999999E+09,8.999999E+09,8.999999E+09,8.999999E+09,8.999999E+09,8.999999E+09]];
    LOCAL CONST Robtarget Tr_meulage_bavure_600 := [[-6.3271142578125,-145.648078125,73.99671875],[0.744033444168216,-0.633100864972437,0.1383814197773,-0.162628753271841],[0,0,0,0],[8.999999E+09,8.999999E+09,8.999999E+09,8.999999E+09,8.999999E+09,8.999999E+09]];
    LOCAL CONST Robtarget Tr_meulage_bavure_601 := [[-8.721798828125,-144.51525,74.050671875],[0.746281690995969,-0.631207505433635,0.136443986700637,-0.161318818684245],[0,0,0,0],[8.999999E+09,8.999999E+09,8.999999E+09,8.999999E+09,8.999999E+09,8.999999E+09]];
    LOCAL CONST Robtarget Tr_meulage_bavure_602 := [[-10.8275166015625,-143.572609375,74.089234375],[0.748751386578802,-0.629998961760244,0.132684142557797,-0.15769460228885],[0,0,0,0],[8.999999E+09,8.999999E+09,8.999999E+09,8.999999E+09,8.999999E+09,8.999999E+09]];
    LOCAL CONST Robtarget Tr_meulage_bavure_603 := [[-12.1863857421875,-142.956125,74.115484375],[0.751467741478203,-0.629518188500758,0.126822631112697,-0.151390568074852],[0,0,0,0],[8.999999E+09,8.999999E+09,8.999999E+09,8.999999E+09,8.999999E+09,8.999999E+09]];
    LOCAL CONST Robtarget Tr_meulage_bavure_604 := [[-14.42857421875,-141.984140625,74.1512890625],[0.754426415830283,-0.62979566236484,0.118510635864632,-0.141962797770634],[0,0,0,0],[8.999999E+09,8.999999E+09,8.999999E+09,8.999999E+09,8.999999E+09,8.999999E+09]];
    LOCAL CONST Robtarget Tr_meulage_bavure_605 := [[-16.45407421875,-141.159140625,74.1748359375],[0.757571445984692,-0.630770208420138,0.107478534576225,-0.12908451883795],[0,0,0,0],[8.999999E+09,8.999999E+09,8.999999E+09,8.999999E+09,8.999999E+09,8.999999E+09]];
    LOCAL CONST Robtarget Tr_meulage_bavure_606 := [[-18.00269140625,-140.54475,74.190125],[0.760719059731795,-0.632287916710494,0.0937658287174766,-0.112811665653878],[0,0,0,0],[8.999999E+09,8.999999E+09,8.999999E+09,8.999999E+09,8.999999E+09,8.999999E+09]];
    LOCAL CONST Robtarget Tr_meulage_bavure_607 := [[-20.13298046875,-139.7688125,74.1996796875],[0.763591418989234,-0.634103911712977,0.0778268678609975,-0.0937195424404925],[0,0,0,0],[8.999999E+09,8.999999E+09,8.999999E+09,8.999999E+09,8.999999E+09,8.999999E+09]];
    LOCAL CONST Robtarget Tr_meulage_bavure_608 := [[-20.90999609375,-139.528203125,74.1961328125],[0.76592181485431,-0.635948885615152,0.0603759782001919,-0.0727154018863705],[0,0,0,0],[8.999999E+09,8.999999E+09,8.999999E+09,8.999999E+09,8.999999E+09,8.999999E+09]];
    LOCAL CONST Robtarget Tr_meulage_bavure_609 := [[-22.09274609375,-139.347203125,74.160015625],[0.767528137239594,-0.637626471985142,0.0420635264029397,-0.050632998290148],[0,0,0,0],[8.999999E+09,8.999999E+09,8.999999E+09,8.999999E+09,8.999999E+09,8.999999E+09]];
    LOCAL CONST Robtarget Tr_meulage_bavure_610 := [[-23.69719921875,-139.24225,74.08771875],[0.768334058967131,-0.639020556085834,0.0231924458699684,-0.0278857165124665],[0,0,0,0],[8.999999E+09,8.999999E+09,8.999999E+09,8.999999E+09,8.999999E+09,8.999999E+09]];
    LOCAL CONST Robtarget Tr_meulage_bavure_611 := [[-24.374802734375,-139.389328125,74.0254453125],[0.768315854264481,-0.640044243712334,0.0037383921006194,-0.00448760526882249],[0,0,0,0],[8.999999E+09,8.999999E+09,8.999999E+09,8.999999E+09,8.999999E+09,8.999999E+09]];
    LOCAL CONST Robtarget Tr_meulage_bavure_612 := [[-25.0231171875,-139.44475,73.9800078125],[0.767447948629461,-0.640617054049295,-0.0161282605180379,0.0193213720604092],[0,0,0,0],[8.999999E+09,8.999999E+09,8.999999E+09,8.999999E+09,8.999999E+09,8.999999E+09]];
    LOCAL CONST Robtarget Tr_meulage_bavure_613 := [[-25.776796875,-139.741125,73.888734375],[0.765797063741848,-0.640697114164267,-0.0355079757262591,0.0424411206940669],[0,0,0,0],[8.999999E+09,8.999999E+09,8.999999E+09,8.999999E+09,8.999999E+09,8.999999E+09]];
    LOCAL CONST Robtarget Tr_meulage_bavure_614 := [[-27.8204140625,-140.40778125,73.6639375],[0.763638090121631,-0.640467249896008,-0.0524370327909535,0.0625214100777687],[0,0,0,0],[8.999999E+09,8.999999E+09,8.999999E+09,8.999999E+09,8.999999E+09,8.999999E+09]];
    LOCAL CONST Robtarget Tr_meulage_bavure_615 := [[-28.256349609375,-140.569109375,73.6128203125],[0.761566769177788,-0.640379284360241,-0.0641340116952044,0.0762709432893699],[0,0,0,0],[8.999999E+09,8.999999E+09,8.999999E+09,8.999999E+09,8.999999E+09,8.999999E+09]];
    LOCAL CONST Robtarget Tr_meulage_bavure_616 := [[-29.77990625,-140.731078125,73.50078125],[0.760319983457932,-0.640993571333073,-0.0677273443998078,0.0803353663385712],[0,0,0,0],[8.999999E+09,8.999999E+09,8.999999E+09,8.999999E+09,8.999999E+09,8.999999E+09]];
    LOCAL CONST Robtarget Tr_meulage_bavure_617 := [[-30.299421875,-140.79353125,73.4613828125],[0.760326494914796,-0.642622463999137,-0.0610343664310596,0.0722135444955984],[0,0,0,0],[8.999999E+09,8.999999E+09,8.999999E+09,8.999999E+09,8.999999E+09,8.999999E+09]];
    LOCAL CONST Robtarget Tr_meulage_bavure_618 := [[-30.5508359375,-140.769953125,73.451234375],[0.761274658118083,-0.644971611523752,-0.043230462969774,0.0510258983955127],[0,0,0,0],[8.999999E+09,8.999999E+09,8.999999E+09,8.999999E+09,8.999999E+09,8.999999E+09]];
    LOCAL CONST Robtarget Tr_meulage_bavure_619 := [[-31.61109765625,-140.618625,73.417046875],[0.762043063646972,-0.647083879224022,-0.0154915544409572,0.0182437424047677],[0,0,0,0],[8.999999E+09,8.999999E+09,8.999999E+09,8.999999E+09,8.999999E+09,8.999999E+09]];
    LOCAL CONST Robtarget Tr_meulage_bavure_620 := [[-32.669583984375,-140.230390625,73.4222421875],[0.761282102618017,-0.647785693389756,0.018594202639625,-0.0218520319705213],[0,0,0,0],[8.999999E+09,8.999999E+09,8.999999E+09,8.999999E+09,8.999999E+09,8.999999E+09]];
    LOCAL CONST Robtarget Tr_meulage_bavure_621 := [[-33.621015625,-139.85071875,73.432],[0.758392549972266,-0.646518407443717,0.0537116350956129,-0.0630059460555852],[0,0,0,0],[8.999999E+09,8.999999E+09,8.999999E+09,8.999999E+09,8.999999E+09,8.999999E+09]];
    LOCAL CONST Robtarget Tr_meulage_bavure_622 := [[-36.0354375,-138.65609375,73.49509375],[0.753967550883944,-0.643777397501476,0.0848725132102082,-0.0993994526226266],[0,0,0,0],[8.999999E+09,8.999999E+09,8.999999E+09,8.999999E+09,8.999999E+09,8.999999E+09]];
    LOCAL CONST Robtarget Tr_meulage_bavure_623 := [[-38.1196875,-137.6063125,73.552625],[0.749249582599206,-0.640612507836876,0.10920778884656,-0.127727587596062],[0,0,0,0],[8.999999E+09,8.999999E+09,8.999999E+09,8.999999E+09,8.999999E+09,8.999999E+09]];
    LOCAL CONST Robtarget Tr_meulage_bavure_624 := [[-38.344984375,-137.490875,73.559171875],[0.745259778584571,-0.637899590212723,0.12621179761913,-0.147453577007357],[0,0,0,0],[8.999999E+09,8.999999E+09,8.999999E+09,8.999999E+09,8.999999E+09,8.999999E+09]];
    LOCAL CONST Robtarget Tr_meulage_bavure_625 := [[-39.4504375,-136.9696875,73.58378125],[0.742417072175826,-0.636004578941579,0.136955215437037,-0.159869745329797],[0,0,0,0],[8.999999E+09,8.999999E+09,8.999999E+09,8.999999E+09,8.999999E+09,8.999999E+09]];
    LOCAL CONST Robtarget Tr_meulage_bavure_626 := [[-41.91994140625,-135.84828125,73.63165625],[0.74066795456292,-0.634891815876617,0.143065066584418,-0.166900419231552],[0,0,0,0],[8.999999E+09,8.999999E+09,8.999999E+09,8.999999E+09,8.999999E+09,8.999999E+09]];
    LOCAL CONST Robtarget Tr_meulage_bavure_627 := [[-44.188953125,-134.74346875,73.687984375],[0.739769667750127,-0.634346020858288,0.146058166156979,-0.170331959998657],[0,0,0,0],[8.999999E+09,8.999999E+09,8.999999E+09,8.999999E+09,8.999999E+09,8.999999E+09]];
    LOCAL CONST Robtarget Tr_meulage_bavure_628 := [[-45.93773046875,-133.907921875,73.72875],[0.739493817221436,-0.63418950786471,0.146946114479787,-0.17134585447241],[0,0,0,0],[8.999999E+09,8.999999E+09,8.999999E+09,8.999999E+09,8.999999E+09,8.999999E+09]];
    !
    !Declaration des points de tronconnage

    !
    !Cycle
    LOCAL PROC Cycle()
        !
        Prise;
        !
        Meulage;
        !
        !
        Depose;
        !
    ENDPROC

    !Trajectoire de prise de la pièce
    LOCAL PROC PRISE()

		!
        !Trigger localisation
        LocalisationPieceTable 707 \model:=1;
        !
        !Approche
		MoveJ Reltool(PicKPosition,0,0,-100),V1000,Z0,Tool_Prehenseur1 \Wobj:=Wobj_vision;
		MoveL Reltool(PicKPosition,0,0,-50),V500,Z0,Tool_Prehenseur1 \Wobj:=Wobj_vision;
		MoveL Reltool(PicKPosition,0,0,-10),V200,Z0,Tool_Prehenseur1 \Wobj:=Wobj_vision;
		MoveL PicKPosition,V100,Fine,Tool_Prehenseur1 \Wobj:=Wobj_vision;

        !Fermeture pince
		Gripper_Close;
        !
		MoveL Reltool(PicKPosition,0,0,-100),V500,Z0,Tool_Prehenseur1 \Wobj:=Wobj_vision;

        !Trigger relocalisation
		LocalisationPiecePrehenseur 707 \model:=1,Ref;
        !
        PEO;
        !
    ENDPROC

    !Trajectoire de tronconnage
    LOCAL PROC Tronconnage()
        !
        !StartMotor1();
        !
        ConfJ \Off;
        ConfL \Off;


    ENDPROC


    !Trajectoire de meulage
    LOCAL PROC Meulage()
        !
        !StartMotor2();
        !

        ConfJ \Off;
        ConfL \Off;


        !---------- Meulage zone : 1 ------------

        !Approche PLAN

        Go_to_Meulage_Plan;
		Tool := ToolOffset(Tool_M1_D500_S0 \Z);

